LIN {X 0,Y 568.212,Z 444.708,A -85,B 0,C 180,E1 26844.426,E2 26844.426} C_VEL
LIN {X 0,Y 568.197,Z 444.71,A -85,B 0,C 180,E1 26841.145,E2 26841.145} C_VEL
LIN {X 0,Y 568.223,Z 444.707,A -85,B 0,C 180,E1 26837.829,E2 26837.829} C_VEL
LIN {X 0,Y 568.203,Z 444.709,A -85,B 0,C 180,E1 26834.47,E2 26834.47} C_VEL
LIN {X 0,Y 568.196,Z 444.71,A -85,B 0,C 180,E1 26831.161,E2 26831.161} C_VEL
LIN {X 0,Y 568.216,Z 444.708,A -85,B 0,C 180,E1 26827.889,E2 26827.889} C_VEL
LIN {X 0,Y 568.195,Z 444.71,A -85,B 0,C 180,E1 26824.542,E2 26824.542} C_VEL
LIN {X 0,Y 568.224,Z 444.705,A -85,B 0,C 180,E1 26821.21,E2 26821.21} C_VEL
LIN {X 0,Y 568.204,Z 444.708,A -85,B 0,C 180,E1 26817.882,E2 26817.882} C_VEL
LIN {X 0,Y 568.202,Z 444.709,A -85,B 0,C 180,E1 26814.648,E2 26814.648} C_VEL
LIN {X 0,Y 568.219,Z 444.706,A -85,B 0,C 180,E1 26811.398,E2 26811.398} C_VEL
LIN {X 0,Y 568.207,Z 444.707,A -85,B 0,C 180,E1 26808.061,E2 26808.061} C_VEL
LIN {X 0,Y 568.224,Z 444.706,A -85,B 0,C 180,E1 26804.636,E2 26804.636} C_VEL
LIN {X 0,Y 568.207,Z 444.707,A -85,B 0,C 180,E1 26801.321,E2 26801.321} C_VEL
LIN {X 0,Y 568.208,Z 444.71,A -85,B 0,C 180,E1 26799.787,E2 26799.787} C_VEL
LIN {X 0,Y 567.184,Z 444.832,A -85,B 0,C 180,E1 26799.011,E2 26799.011} C_VEL
LIN {X 0,Y 560.815,Z 445.632,A -85,B 0,C 180,E1 26796.831,E2 26796.831} C_VEL
LIN {X 0,Y 560.283,Z 445.694,A -85,B 0,C 180,E1 26796.264,E2 26796.264} C_VEL
LIN {X 0,Y 560.263,Z 445.695,A -85,B 0,C 180,E1 26792.93,E2 26792.93} C_VEL
LIN {X 0,Y 560.252,Z 445.696,A -85,B 0,C 180,E1 26789.665,E2 26789.665} C_VEL
LIN {X 0,Y 560.278,Z 445.695,A -85,B 0,C 180,E1 26786.412,E2 26786.412} C_VEL
LIN {X 0,Y 560.262,Z 445.697,A -85,B 0,C 180,E1 26783.083,E2 26783.083} C_VEL
LIN {X 0,Y 560.286,Z 445.693,A -85,B 0,C 180,E1 26779.759,E2 26779.759} C_VEL
LIN {X 0,Y 560.269,Z 445.697,A -85,B 0,C 180,E1 26776.431,E2 26776.431} C_VEL
LIN {X 0,Y 560.255,Z 445.701,A -85,B 0,C 180,E1 26773.119,E2 26773.119} C_VEL
LIN {X 0,Y 560.278,Z 445.696,A -85,B 0,C 180,E1 26769.882,E2 26769.882} C_VEL
LIN {X 0,Y 560.269,Z 445.7,A -85,B 0,C 180,E1 26766.575,E2 26766.575} C_VEL
LIN {X 0,Y 560.238,Z 445.797,A -85,B 0,C 180,E1 26764.175,E2 26764.175} C_VEL
LIN {X 0,Y 564.833,Z 458.966,A -85,B 0,C 180,E1 26762.797,E2 26762.797} C_VEL
LIN {X 0,Y 564.124,Z 495.402,A -85,B 0,C 180,E1 26759.984,E2 26759.984} C_VEL
LIN {X 0,Y 565.707,Z 504.661,A -85,B 0,C 180,E1 26759.758,E2 26759.758} C_VEL
LIN {X 0,Y 564.489,Z 747.125,A -85,B 0,C 180,E1 26756.4,E2 26756.4} C_VEL
LIN {X 0,Y 564.25,Z 768.15,A -85,B 0,C 180,E1 26755.998,E2 26755.998} C_VEL
LIN {X 0,Y 563.894,Z 788.378,A -85,B 0,C 180,E1 26755.42,E2 26755.42} C_VEL
LIN {X 0,Y 563.454,Z 808.539,A -85,B 0,C 180,E1 26754.645,E2 26754.645} C_VEL
LIN {X 0,Y 562.959,Z 828.494,A -85,B 0,C 180,E1 26753.665,E2 26753.665} C_VEL
LIN {X 0,Y 562.466,Z 847.374,A -85,B 0,C 180,E1 26752.519,E2 26752.519} C_VEL
LIN {X 0,Y 561.985,Z 864.434,A -85,B 0,C 180,E1 26751.281,E2 26751.281} C_VEL
LIN {X 0,Y 561.503,Z 881.299,A -85,B 0,C 180,E1 26749.829,E2 26749.829} C_VEL
LIN {X 0,Y 561.07,Z 897.052,A -85,B 0,C 180,E1 26748.224,E2 26748.224} C_VEL
LIN {X 0,Y 560.702,Z 911.608,A -85,B 0,C 180,E1 26746.471,E2 26746.471} C_VEL
LIN {X 0,Y 560.418,Z 924.193,A -85,B 0,C 180,E1 26744.675,E2 26744.675} C_VEL
LIN {X 0,Y 560.211,Z 935.329,A -85,B 0,C 180,E1 26742.786,E2 26742.786} C_VEL
LIN {X 0,Y 560.059,Z 944.99,A -85,B 0,C 180,E1 26740.804,E2 26740.804} C_VEL
LIN {X 0,Y 559.979,Z 953.12,A -85,B 0,C 180,E1 26738.729,E2 26738.729} C_VEL
LIN {X 0,Y 559.94,Z 959.122,A -85,B 0,C 180,E1 26736.768,E2 26736.768} C_VEL
LIN {X 0,Y 559.919,Z 963.693,A -85,B 0,C 180,E1 26734.711,E2 26734.711} C_VEL
LIN {X 0,Y 559.912,Z 966.567,A -85,B 0,C 180,E1 26732.661,E2 26732.661} C_VEL
LIN {X 0,Y 559.902,Z 967.886,A -85,B 0,C 180,E1 26730.511,E2 26730.511} C_VEL
LIN {X 0,Y 559.901,Z 967.469,A -85,B 0,C 180,E1 26728.362,E2 26728.362} C_VEL
LIN {X 0,Y 559.908,Z 965.467,A -85,B 0,C 180,E1 26726.314,E2 26726.314} C_VEL
LIN {X 0,Y 559.924,Z 961.822,A -85,B 0,C 180,E1 26724.26,E2 26724.26} C_VEL
LIN {X 0,Y 559.958,Z 956.427,A -85,B 0,C 180,E1 26722.2,E2 26722.2} C_VEL
LIN {X 0,Y 560.011,Z 949.242,A -85,B 0,C 180,E1 26720.13,E2 26720.13} C_VEL
LIN {X 0,Y 560.118,Z 940.592,A -85,B 0,C 180,E1 26718.153,E2 26718.153} C_VEL
LIN {X 0,Y 560.29,Z 930.551,A -85,B 0,C 180,E1 26716.27,E2 26716.27} C_VEL
LIN {X 0,Y 560.546,Z 918.433,A -85,B 0,C 180,E1 26714.374,E2 26714.374} C_VEL
LIN {X 0,Y 560.872,Z 904.72,A -85,B 0,C 180,E1 26712.572,E2 26712.572} C_VEL
LIN {X 0,Y 561.284,Z 889.331,A -85,B 0,C 180,E1 26710.866,E2 26710.866} C_VEL
LIN {X 0,Y 561.752,Z 872.597,A -85,B 0,C 180,E1 26709.3,E2 26709.3} C_VEL
LIN {X 0,Y 562.239,Z 855.595,A -85,B 0,C 180,E1 26707.961,E2 26707.961} C_VEL
LIN {X 0,Y 562.736,Z 837.569,A -85,B 0,C 180,E1 26706.768,E2 26706.768} C_VEL
LIN {X 0,Y 563.217,Z 818.644,A -85,B 0,C 180,E1 26705.733,E2 26705.733} C_VEL
LIN {X 0,Y 563.681,Z 798.675,A -85,B 0,C 180,E1 26704.86,E2 26704.86} C_VEL
LIN {X 0,Y 564.083,Z 778.165,A -85,B 0,C 180,E1 26704.174,E2 26704.174} C_VEL
LIN {X 0,Y 564.386,Z 757.733,A -85,B 0,C 180,E1 26703.688,E2 26703.688} C_VEL
LIN {X 0,Y 564.677,Z 708.736,A -85,B 0,C 180,E1 26702.983,E2 26702.983} C_VEL
LIN {X 0,Y 565.566,Z 507.584,A -85,B 0,C 180,E1 26700.186,E2 26700.186} C_VEL
LIN {X 0,Y 562.933,Z 497.494,A -85,B 0,C 180,E1 26699.882,E2 26699.882} C_VEL
LIN {X 0,Y 563.492,Z 471.301,A -85,B 0,C 180,E1 26696.81,E2 26696.81} C_VEL
LIN {X 0,Y 563.723,Z 457.22,A -85,B 0,C 180,E1 26695.118,E2 26695.118} C_VEL
LIN {X 0,Y 560.258,Z 445.701,A -85,B 0,C 180,E1 26693.474,E2 26693.474} C_VEL
LIN {X 0,Y 560.243,Z 445.699,A -85,B 0,C 180,E1 26690.123,E2 26690.123} C_VEL
LIN {X 0,Y 560.278,Z 445.693,A -85,B 0,C 180,E1 26686.878,E2 26686.878} C_VEL
LIN {X 0,Y 560.261,Z 445.695,A -85,B 0,C 180,E1 26683.541,E2 26683.541} C_VEL
LIN {X 0,Y 560.269,Z 445.691,A -85,B 0,C 180,E1 26680.109,E2 26680.109} C_VEL
LIN {X 0,Y 560.268,Z 445.697,A -85,B 0,C 180,E1 26676.843,E2 26676.843} C_VEL
LIN {X 0,Y 560.272,Z 445.699,A -85,B 0,C 180,E1 26673.466,E2 26673.466} C_VEL
LIN {X 0,Y 560.282,Z 445.696,A -85,B 0,C 180,E1 26670.058,E2 26670.058} C_VEL
LIN {X 0,Y 560.296,Z 445.883,A -85,B 0,C 180,E1 26668.994,E2 26668.994} C_VEL
LIN {X 0,Y 564.194,Z 457.95,A -85,B 0,C 180,E1 26667.551,E2 26667.551} C_VEL
LIN {X 0,Y 563.64,Z 489.328,A -85,B 0,C 180,E1 26664.582,E2 26664.582} C_VEL
LIN {X 0,Y 562.831,Z 522.784,A -85,B 0,C 180,E1 26661.467,E2 26661.467} C_VEL
LIN {X 0,Y 562.016,Z 560.717,A -85,B 0,C 180,E1 26657.979,E2 26657.979} C_VEL
LIN {X 0,Y 561.307,Z 595.844,A -85,B 0,C 180,E1 26654.758,E2 26654.758} C_VEL
LIN {X 0,Y 561.234,Z 603.069,A -85,B 0,C 180,E1 26654.135,E2 26654.135} C_VEL
LIN {X 0,Y 561.827,Z 610.203,A -85,B 0,C 180,E1 26654.019,E2 26654.019} C_VEL
LIN {X 0,Y 561.418,Z 743.182,A -85,B 0,C 180,E1 26652.262,E2 26652.262} C_VEL
LIN {X 0,Y 561.293,Z 759.345,A -85,B 0,C 180,E1 26651.88,E2 26651.88} C_VEL
LIN {X 0,Y 561.125,Z 773.652,A -85,B 0,C 180,E1 26651.356,E2 26651.356} C_VEL
LIN {X 0,Y 560.927,Z 786.575,A -85,B 0,C 180,E1 26650.735,E2 26650.735} C_VEL
LIN {X 0,Y 560.744,Z 799.431,A -85,B 0,C 180,E1 26649.96,E2 26649.96} C_VEL
LIN {X 0,Y 560.515,Z 813.552,A -85,B 0,C 180,E1 26648.876,E2 26648.876} C_VEL
LIN {X 0,Y 560.345,Z 823.86,A -85,B 0,C 180,E1 26647.897,E2 26647.897} C_VEL
LIN {X 0,Y 560.199,Z 833.784,A -85,B 0,C 180,E1 26646.765,E2 26646.765} C_VEL
LIN {X 0,Y 560.07,Z 843.961,A -85,B 0,C 180,E1 26645.327,E2 26645.327} C_VEL
LIN {X 0,Y 559.99,Z 851.364,A -85,B 0,C 180,E1 26643.993,E2 26643.993} C_VEL
LIN {X 0,Y 559.947,Z 857.668,A -85,B 0,C 180,E1 26642.559,E2 26642.559} C_VEL
LIN {X 0,Y 559.924,Z 863.148,A -85,B 0,C 180,E1 26640.819,E2 26640.819} C_VEL
LIN {X 0,Y 559.915,Z 866.195,A -85,B 0,C 180,E1 26639.284,E2 26639.284} C_VEL
LIN {X 0,Y 559.913,Z 867.841,A -85,B 0,C 180,E1 26637.646,E2 26637.646} C_VEL
LIN {X 0,Y 559.913,Z 867.666,A -85,B 0,C 180,E1 26636.007,E2 26636.007} C_VEL
LIN {X 0,Y 559.918,Z 865.949,A -85,B 0,C 180,E1 26634.467,E2 26634.467} C_VEL
LIN {X 0,Y 559.923,Z 862.739,A -85,B 0,C 180,E1 26632.923,E2 26632.923} C_VEL
LIN {X 0,Y 559.947,Z 857.342,A -85,B 0,C 180,E1 26631.27,E2 26631.27} C_VEL
LIN {X 0,Y 559.991,Z 851.393,A -85,B 0,C 180,E1 26629.923,E2 26629.923} C_VEL
LIN {X 0,Y 560.083,Z 843.245,A -85,B 0,C 180,E1 26628.467,E2 26628.467} C_VEL
LIN {X 0,Y 560.202,Z 833.489,A -85,B 0,C 180,E1 26627.109,E2 26627.109} C_VEL
LIN {X 0,Y 560.345,Z 823.82,A -85,B 0,C 180,E1 26626.008,E2 26626.008} C_VEL
LIN {X 0,Y 560.545,Z 812.105,A -85,B 0,C 180,E1 26624.905,E2 26624.905} C_VEL
LIN {X 0,Y 560.748,Z 798.703,A -85,B 0,C 180,E1 26623.903,E2 26623.903} C_VEL
LIN {X 0,Y 560.936,Z 786.019,A -85,B 0,C 180,E1 26623.145,E2 26623.145} C_VEL
LIN {X 0,Y 561.137,Z 773.052,A -85,B 0,C 180,E1 26622.528,E2 26622.528} C_VEL
LIN {X 0,Y 561.312,Z 756.063,A -85,B 0,C 180,E1 26621.941,E2 26621.941} C_VEL
LIN {X 0,Y 561.419,Z 741.983,A -85,B 0,C 180,E1 26621.627,E2 26621.627} C_VEL
LIN {X 0,Y 561.632,Z 605.827,A -85,B 0,C 180,E1 26619.816,E2 26619.816} C_VEL
LIN {X 0,Y 561.436,Z 603.897,A -85,B 0,C 180,E1 26619.761,E2 26619.761} C_VEL
LIN {X 0,Y 562.877,Z 569.056,A -85,B 0,C 180,E1 26616.387,E2 26616.387} C_VEL
LIN {X 0,Y 564.91,Z 533.555,A -85,B 0,C 180,E1 26612.829,E2 26612.829} C_VEL
LIN {X 0,Y 567.601,Z 501.05,A -85,B 0,C 180,E1 26609.397,E2 26609.397} C_VEL
LIN {X 0,Y 569.345,Z 484.628,A -85,B 0,C 180,E1 26607.554,E2 26607.554} C_VEL
LIN {X 0,Y 570.786,Z 468.2,A -85,B 0,C 180,E1 26605.475,E2 26605.475} C_VEL
LIN {X 0,Y 568.716,Z 463.182,A -85,B 0,C 180,E1 26604.29,E2 26604.29} C_VEL
LIN {X 0,Y 567.301,Z 459.69,A -85,B 0,C 180,E1 26603.31,E2 26603.31} C_VEL
LIN {X 0,Y 565.739,Z 455.845,A -85,B 0,C 180,E1 26601.858,E2 26601.858} C_VEL
LIN {X 0,Y 564.732,Z 454.619,A -85,B 0,C 180,E1 26600.529,E2 26600.529} C_VEL
LIN {X 0,Y 564.984,Z 454.894,A -85,B 0,C 180,E1 26599.364,E2 26599.364} C_VEL
LIN {X 0,Y 566.259,Z 456.589,A -85,B 0,C 180,E1 26598.324,E2 26598.324} C_VEL
LIN {X 0,Y 567.907,Z 460.494,A -85,B 0,C 180,E1 26597.326,E2 26597.326} C_VEL
LIN {X 0,Y 569.112,Z 464.051,A -85,B 0,C 180,E1 26596.71,E2 26596.71} C_VEL
LIN {X 0,Y 566.813,Z 482.57,A -85,B 0,C 180,E1 26595.237,E2 26595.237} C_VEL
LIN {X 0,Y 564.922,Z 510.213,A -85,B 0,C 180,E1 26593.302,E2 26593.302} C_VEL
LIN {X 0,Y 564.287,Z 540.963,A -85,B 0,C 180,E1 26591.298,E2 26591.298} C_VEL
LIN {X 0,Y 565.775,Z 557.767,A -85,B 0,C 180,E1 26590.169,E2 26590.169} C_VEL
LIN {X 0,Y 568.608,Z 569.698,A -85,B 0,C 180,E1 26589.312,E2 26589.312} C_VEL
LIN {X 0,Y 572.485,Z 578.868,A -85,B 0,C 180,E1 26588.596,E2 26588.596} C_VEL
LIN {X 0,Y 577.865,Z 586.598,A -85,B 0,C 180,E1 26587.908,E2 26587.908} C_VEL
LIN {X 0,Y 583.498,Z 591.893,A -85,B 0,C 180,E1 26587.336,E2 26587.336} C_VEL
LIN {X 0,Y 587.347,Z 594.24,A -85,B 0,C 180,E1 26586.861,E2 26586.861} C_VEL
LIN {X 0,Y 590.651,Z 595.228,A -85,B 0,C 180,E1 26586.315,E2 26586.315} C_VEL
LIN {X 0,Y 592.846,Z 594.931,A -85,B 0,C 180,E1 26585.784,E2 26585.784} C_VEL
LIN {X 0,Y 594.074,Z 593.569,A -85,B 0,C 180,E1 26585.261,E2 26585.261} C_VEL
LIN {X 0,Y 594.221,Z 590.934,A -85,B 0,C 180,E1 26584.692,E2 26584.692} C_VEL
LIN {X 0,Y 592.942,Z 587.105,A -85,B 0,C 180,E1 26584.162,E2 26584.162} C_VEL
LIN {X 0,Y 589.902,Z 581.364,A -85,B 0,C 180,E1 26583.66,E2 26583.66} C_VEL
LIN {X 0,Y 586.325,Z 572.675,A -85,B 0,C 180,E1 26583.131,E2 26583.131} C_VEL
LIN {X 0,Y 583.607,Z 562.507,A -85,B 0,C 180,E1 26582.72,E2 26582.72} C_VEL
LIN {X 0,Y 581.84,Z 551.15,A -85,B 0,C 180,E1 26582.448,E2 26582.448} C_VEL
LIN {X 0,Y 580.983,Z 537.863,A -85,B 0,C 180,E1 26582.315,E2 26582.315} C_VEL
LIN {X 0,Y 580.854,Z 522.497,A -85,B 0,C 180,E1 26582.295,E2 26582.295} C_VEL
LIN {X 0,Y 577.341,Z 528.82,A -85,B 0,C 180,E1 26581.739,E2 26581.739} C_VEL
LIN {X 0,Y 574.597,Z 531.681,A -85,B 0,C 180,E1 26581.294,E2 26581.294} C_VEL
LIN {X 0,Y 569.784,Z 544.591,A -85,B 0,C 180,E1 26580.489,E2 26580.489} C_VEL
LIN {X 0,Y 568.425,Z 548.114,A -85,B 0,C 180,E1 26580.255,E2 26580.255} C_VEL
LIN {X 0,Y 567.076,Z 552.625,A -85,B 0,C 180,E1 26580.021,E2 26580.021} C_VEL
LIN {X 0,Y 565.954,Z 557.205,A -85,B 0,C 180,E1 26579.823,E2 26579.823} C_VEL
LIN {X 0,Y 565.633,Z 557.842,A -85,B 0,C 180,E1 26579.762,E2 26579.762} C_VEL
LIN {X 0,Y 564.41,Z 806.369,A -85,B 0,C 180,E1 26576.292,E2 26576.292} C_VEL
LIN {X 0,Y 564.094,Z 827.689,A -85,B 0,C 180,E1 26575.795,E2 26575.795} C_VEL
LIN {X 0,Y 563.708,Z 847.582,A -85,B 0,C 180,E1 26575.139,E2 26575.139} C_VEL
LIN {X 0,Y 563.277,Z 866.639,A -85,B 0,C 180,E1 26574.32,E2 26574.32} C_VEL
LIN {X 0,Y 562.788,Z 885.877,A -85,B 0,C 180,E1 26573.291,E2 26573.291} C_VEL
LIN {X 0,Y 562.289,Z 903.978,A -85,B 0,C 180,E1 26572.114,E2 26572.114} C_VEL
LIN {X 0,Y 561.774,Z 921.539,A -85,B 0,C 180,E1 26570.744,E2 26570.744} C_VEL
LIN {X 0,Y 561.289,Z 938.854,A -85,B 0,C 180,E1 26569.134,E2 26569.134} C_VEL
LIN {X 0,Y 560.896,Z 953.414,A -85,B 0,C 180,E1 26567.534,E2 26567.534} C_VEL
LIN {X 0,Y 560.564,Z 967.357,A -85,B 0,C 180,E1 26565.731,E2 26565.731} C_VEL
LIN {X 0,Y 560.314,Z 979.299,A -85,B 0,C 180,E1 26563.893,E2 26563.893} C_VEL
LIN {X 0,Y 560.132,Z 989.854,A -85,B 0,C 180,E1 26561.951,E2 26561.951} C_VEL
LIN {X 0,Y 560.016,Z 998.675,A -85,B 0,C 180,E1 26559.974,E2 26559.974} C_VEL
LIN {X 0,Y 559.958,Z 1005.979,A -85,B 0,C 180,E1 26557.903,E2 26557.903} C_VEL
LIN {X 0,Y 559.93,Z 1011.245,A -85,B 0,C 180,E1 26555.944,E2 26555.944} C_VEL
LIN {X 0,Y 559.915,Z 1015.258,A -85,B 0,C 180,E1 26553.789,E2 26553.789} C_VEL
LIN {X 0,Y 559.907,Z 1017.386,A -85,B 0,C 180,E1 26551.74,E2 26551.74} C_VEL
LIN {X 0,Y 559.9,Z 1017.918,A -85,B 0,C 180,E1 26549.591,E2 26549.591} C_VEL
LIN {X 0,Y 559.907,Z 1016.847,A -85,B 0,C 180,E1 26547.544,E2 26547.544} C_VEL
LIN {X 0,Y 559.917,Z 1013.957,A -85,B 0,C 180,E1 26545.391,E2 26545.391} C_VEL
LIN {X 0,Y 559.937,Z 1009.727,A -85,B 0,C 180,E1 26543.438,E2 26543.438} C_VEL
LIN {X 0,Y 559.979,Z 1003.64,A -85,B 0,C 180,E1 26541.375,E2 26541.375} C_VEL
LIN {X 0,Y 560.052,Z 996.107,A -85,B 0,C 180,E1 26539.404,E2 26539.404} C_VEL
LIN {X 0,Y 560.195,Z 986.708,A -85,B 0,C 180,E1 26537.424,E2 26537.424} C_VEL
LIN {X 0,Y 560.381,Z 975.799,A -85,B 0,C 180,E1 26535.535,E2 26535.535} C_VEL
LIN {X 0,Y 560.681,Z 962.62,A -85,B 0,C 180,E1 26533.619,E2 26533.619} C_VEL
LIN {X 0,Y 561.017,Z 948.816,A -85,B 0,C 180,E1 26531.935,E2 26531.935} C_VEL
LIN {X 0,Y 561.46,Z 932.865,A -85,B 0,C 180,E1 26530.278,E2 26530.278} C_VEL
LIN {X 0,Y 561.94,Z 916.056,A -85,B 0,C 180,E1 26528.804,E2 26528.804} C_VEL
LIN {X 0,Y 562.446,Z 898.096,A -85,B 0,C 180,E1 26527.482,E2 26527.482} C_VEL
LIN {X 0,Y 562.937,Z 879.326,A -85,B 0,C 180,E1 26526.334,E2 26526.334} C_VEL
LIN {X 0,Y 563.439,Z 859.599,A -85,B 0,C 180,E1 26525.354,E2 26525.354} C_VEL
LIN {X 0,Y 563.895,Z 839.169,A -85,B 0,C 180,E1 26524.559,E2 26524.559} C_VEL
LIN {X 0,Y 564.243,Z 818.543,A -85,B 0,C 180,E1 26523.966,E2 26523.966} C_VEL
LIN {X 0,Y 564.48,Z 797.161,A -85,B 0,C 180,E1 26523.557,E2 26523.557} C_VEL
LIN {X 0,Y 565.701,Z 557.499,A -85,B 0,C 180,E1 26520.221,E2 26520.221} C_VEL
LIN {X 0,Y 566.509,Z 555.474,A -85,B 0,C 180,E1 26520.079,E2 26520.079} C_VEL
LIN {X 0,Y 567.509,Z 551.007,A -85,B 0,C 180,E1 26519.904,E2 26519.904} C_VEL
LIN {X 0,Y 569.272,Z 545.742,A -85,B 0,C 180,E1 26519.599,E2 26519.599} C_VEL
LIN {X 0,Y 573.361,Z 535.153,A -85,B 0,C 180,E1 26518.91,E2 26518.91} C_VEL
LIN {X 0,Y 574.591,Z 531.68,A -85,B 0,C 180,E1 26518.707,E2 26518.707} C_VEL
LIN {X 0,Y 577.335,Z 528.827,A -85,B 0,C 180,E1 26518.262,E2 26518.262} C_VEL
LIN {X 0,Y 580.897,Z 522.403,A -85,B 0,C 180,E1 26517.698,E2 26517.698} C_VEL
LIN {X 0,Y 581.148,Z 542.214,A -85,B 0,C 180,E1 26517.659,E2 26517.659} C_VEL
LIN {X 0,Y 582.272,Z 554.667,A -85,B 0,C 180,E1 26517.485,E2 26517.485} C_VEL
LIN {X 0,Y 584.278,Z 565.498,A -85,B 0,C 180,E1 26517.178,E2 26517.178} C_VEL
LIN {X 0,Y 587.14,Z 574.973,A -85,B 0,C 180,E1 26516.747,E2 26516.747} C_VEL
LIN {X 0,Y 590.798,Z 583.078,A -85,B 0,C 180,E1 26516.21,E2 26516.21} C_VEL
LIN {X 0,Y 593.208,Z 587.704,A -85,B 0,C 180,E1 26515.769,E2 26515.769} C_VEL
LIN {X 0,Y 594.283,Z 591.409,A -85,B 0,C 180,E1 26515.226,E2 26515.226} C_VEL
LIN {X 0,Y 594.044,Z 593.64,A -85,B 0,C 180,E1 26514.718,E2 26514.718} C_VEL
LIN {X 0,Y 592.459,Z 595.083,A -85,B 0,C 180,E1 26514.102,E2 26514.102} C_VEL
LIN {X 0,Y 589.617,Z 595.055,A -85,B 0,C 180,E1 26513.494,E2 26513.494} C_VEL
LIN {X 0,Y 586.119,Z 593.612,A -85,B 0,C 180,E1 26512.973,E2 26512.973} C_VEL
LIN {X 0,Y 580.24,Z 589.13,A -85,B 0,C 180,E1 26512.273,E2 26512.273} C_VEL
LIN {X 0,Y 575.058,Z 582.688,A -85,B 0,C 180,E1 26511.505,E2 26511.505} C_VEL
LIN {X 0,Y 571.39,Z 575.079,A -85,B 0,C 180,E1 26510.743,E2 26510.743} C_VEL
LIN {X 0,Y 568.573,Z 564.258,A -85,B 0,C 180,E1 26509.806,E2 26509.806} C_VEL
LIN {X 0,Y 567.205,Z 550.519,A -85,B 0,C 180,E1 26508.756,E2 26508.756} C_VEL
LIN {X 0,Y 568.262,Z 497.326,A -85,B 0,C 180,E1 26504.983,E2 26504.983} C_VEL
LIN {X 0,Y 569.217,Z 464.903,A -85,B 0,C 180,E1 26502.585,E2 26502.585} C_VEL
LIN {X 0,Y 561.938,Z 449.676,A -85,B 0,C 180,E1 26500.634,E2 26500.634} C_VEL
LIN {X 0,Y 560.368,Z 446.244,A -85,B 0,C 180,E1 26500.187,E2 26500.187} C_VEL
LIN {X 0,Y 560.28,Z 445.7,A -85,B 0,C 180,E1 26500.108,E2 26500.108} C_VEL
LIN {X 0,Y 560.229,Z 445.698,A -85,B 0,C 180,E1 26496.913,E2 26496.913} C_VEL
LIN {X 0,Y 560.258,Z 445.696,A -85,B 0,C 180,E1 26493.549,E2 26493.549} C_VEL
LIN {X 0,Y 560.259,Z 445.696,A -85,B 0,C 180,E1 26490.335,E2 26490.335} C_VEL
LIN {X 0,Y 560.233,Z 445.699,A -85,B 0,C 180,E1 26486.957,E2 26486.957} C_VEL
LIN {X 0,Y 560.28,Z 445.693,A -85,B 0,C 180,E1 26483.674,E2 26483.674} C_VEL
LIN {X 0,Y 560.225,Z 445.699,A -85,B 0,C 180,E1 26480.449,E2 26480.449} C_VEL
LIN {X 0,Y 560.255,Z 445.696,A -85,B 0,C 180,E1 26477.018,E2 26477.018} C_VEL
LIN {X 0,Y 560.257,Z 445.696,A -85,B 0,C 180,E1 26473.836,E2 26473.836} C_VEL
LIN {X 0,Y 560.227,Z 445.699,A -85,B 0,C 180,E1 26470.46,E2 26470.46} C_VEL
LIN {X 0,Y 560.281,Z 445.692,A -85,B 0,C 180,E1 26467.156,E2 26467.156} C_VEL
LIN {X 0,Y 560.225,Z 445.699,A -85,B 0,C 180,E1 26463.918,E2 26463.918} C_VEL
LIN {X 0,Y 560.253,Z 445.695,A -85,B 0,C 180,E1 26460.511,E2 26460.511} C_VEL
LIN {X 0,Y 560.256,Z 445.695,A -85,B 0,C 180,E1 26457.34,E2 26457.34} C_VEL
LIN {X 0,Y 560.225,Z 445.698,A -85,B 0,C 180,E1 26453.955,E2 26453.955} C_VEL
LIN {X 0,Y 560.279,Z 445.691,A -85,B 0,C 180,E1 26450.701,E2 26450.701} C_VEL
LIN {X 0,Y 560.228,Z 445.695,A -85,B 0,C 180,E1 26447.424,E2 26447.424} C_VEL
LIN {X 0,Y 560.251,Z 445.696,A -85,B 0,C 180,E1 26443.941,E2 26443.941} C_VEL
LIN {X 0,Y 560.26,Z 445.693,A -85,B 0,C 180,E1 26440.722,E2 26440.722} C_VEL
LIN {X 0,Y 560.225,Z 445.694,A -85,B 0,C 180,E1 26437.324,E2 26437.324} C_VEL
LIN {X 0,Y 560.283,Z 445.694,A -85,B 0,C 180,E1 26436.264,E2 26436.264} C_VEL
LIN {X 0,Y 559.284,Z 445.817,A -85,B 0,C 180,E1 26435.476,E2 26435.476} C_VEL
LIN {X 0,Y 552.853,Z 446.619,A -85,B 0,C 180,E1 26433.265,E2 26433.265} C_VEL
LIN {X 0,Y 552.32,Z 446.682,A -85,B 0,C 180,E1 26432.689,E2 26432.689} C_VEL
LIN {X 0,Y 552.289,Z 446.685,A -85,B 0,C 180,E1 26429.301,E2 26429.301} C_VEL
LIN {X 0,Y 552.339,Z 446.681,A -85,B 0,C 180,E1 26426.113,E2 26426.113} C_VEL
LIN {X 0,Y 552.301,Z 446.686,A -85,B 0,C 180,E1 26422.796,E2 26422.796} C_VEL
LIN {X 0,Y 552.328,Z 446.681,A -85,B 0,C 180,E1 26419.467,E2 26419.467} C_VEL
LIN {X 0,Y 552.323,Z 446.686,A -85,B 0,C 180,E1 26416.244,E2 26416.244} C_VEL
LIN {X 0,Y 552.298,Z 446.69,A -85,B 0,C 180,E1 26412.897,E2 26412.897} C_VEL
LIN {X 0,Y 552.339,Z 446.684,A -85,B 0,C 180,E1 26409.705,E2 26409.705} C_VEL
LIN {X 0,Y 552.307,Z 446.69,A -85,B 0,C 180,E1 26406.297,E2 26406.297} C_VEL
LIN {X 0,Y 552.311,Z 446.756,A -85,B 0,C 180,E1 26404.641,E2 26404.641} C_VEL
LIN {X 0,Y 557.679,Z 461.976,A -85,B 0,C 180,E1 26403.027,E2 26403.027} C_VEL
LIN {X 0,Y 556.92,Z 495.437,A -85,B 0,C 180,E1 26400.412,E2 26400.412} C_VEL
LIN {X 0,Y 558.758,Z 505.983,A -85,B 0,C 180,E1 26400.148,E2 26400.148} C_VEL
LIN {X 0,Y 557.305,Z 748.805,A -85,B 0,C 180,E1 26396.741,E2 26396.741} C_VEL
LIN {X 0,Y 557.019,Z 769.975,A -85,B 0,C 180,E1 26396.318,E2 26396.318} C_VEL
LIN {X 0,Y 556.593,Z 790.574,A -85,B 0,C 180,E1 26395.703,E2 26395.703} C_VEL
LIN {X 0,Y 556.085,Z 809.793,A -85,B 0,C 180,E1 26394.937,E2 26394.937} C_VEL
LIN {X 0,Y 555.518,Z 829.135,A -85,B 0,C 180,E1 26393.965,E2 26393.965} C_VEL
LIN {X 0,Y 554.928,Z 848.12,A -85,B 0,C 180,E1 26392.791,E2 26392.791} C_VEL
LIN {X 0,Y 554.335,Z 865.766,A -85,B 0,C 180,E1 26391.478,E2 26391.478} C_VEL
LIN {X 0,Y 553.789,Z 881.86,A -85,B 0,C 180,E1 26390.062,E2 26390.062} C_VEL
LIN {X 0,Y 553.279,Z 897.649,A -85,B 0,C 180,E1 26388.422,E2 26388.422} C_VEL
LIN {X 0,Y 552.857,Z 911.61,A -85,B 0,C 180,E1 26386.711,E2 26386.711} C_VEL
LIN {X 0,Y 552.524,Z 924.195,A -85,B 0,C 180,E1 26384.89,E2 26384.89} C_VEL
LIN {X 0,Y 552.274,Z 935.33,A -85,B 0,C 180,E1 26382.973,E2 26382.973} C_VEL
LIN {X 0,Y 552.093,Z 944.995,A -85,B 0,C 180,E1 26380.961,E2 26380.961} C_VEL
LIN {X 0,Y 551.989,Z 953.123,A -85,B 0,C 180,E1 26378.856,E2 26378.856} C_VEL
LIN {X 0,Y 551.94,Z 959.125,A -85,B 0,C 180,E1 26376.866,E2 26376.866} C_VEL
LIN {X 0,Y 551.92,Z 963.695,A -85,B 0,C 180,E1 26374.78,E2 26374.78} C_VEL
LIN {X 0,Y 551.913,Z 966.568,A -85,B 0,C 180,E1 26372.699,E2 26372.699} C_VEL
LIN {X 0,Y 551.902,Z 967.886,A -85,B 0,C 180,E1 26370.518,E2 26370.518} C_VEL
LIN {X 0,Y 551.902,Z 967.469,A -85,B 0,C 180,E1 26368.338,E2 26368.338} C_VEL
LIN {X 0,Y 551.91,Z 965.466,A -85,B 0,C 180,E1 26366.26,E2 26366.26} C_VEL
LIN {X 0,Y 551.929,Z 961.821,A -85,B 0,C 180,E1 26364.177,E2 26364.177} C_VEL
LIN {X 0,Y 551.965,Z 956.426,A -85,B 0,C 180,E1 26362.086,E2 26362.086} C_VEL
LIN {X 0,Y 552.033,Z 949.241,A -85,B 0,C 180,E1 26359.986,E2 26359.986} C_VEL
LIN {X 0,Y 552.177,Z 940.076,A -85,B 0,C 180,E1 26357.874,E2 26357.874} C_VEL
LIN {X 0,Y 552.401,Z 929.287,A -85,B 0,C 180,E1 26355.856,E2 26355.856} C_VEL
LIN {X 0,Y 552.709,Z 916.902,A -85,B 0,C 180,E1 26353.931,E2 26353.931} C_VEL
LIN {X 0,Y 553.087,Z 903.805,A -85,B 0,C 180,E1 26352.21,E2 26352.21} C_VEL
LIN {X 0,Y 553.568,Z 888.801,A -85,B 0,C 180,E1 26350.535,E2 26350.535} C_VEL
LIN {X 0,Y 554.12,Z 872.076,A -85,B 0,C 180,E1 26348.956,E2 26348.956} C_VEL
LIN {X 0,Y 554.734,Z 854.133,A -85,B 0,C 180,E1 26347.535,E2 26347.535} C_VEL
LIN {X 0,Y 555.33,Z 835.779,A -85,B 0,C 180,E1 26346.327,E2 26346.327} C_VEL
LIN {X 0,Y 555.905,Z 816.826,A -85,B 0,C 180,E1 26345.301,E2 26345.301} C_VEL
LIN {X 0,Y 556.431,Z 796.657,A -85,B 0,C 180,E1 26344.429,E2 26344.429} C_VEL
LIN {X 0,Y 556.882,Z 776.082,A -85,B 0,C 180,E1 26343.756,E2 26343.756} C_VEL
LIN {X 0,Y 557.241,Z 754.862,A -85,B 0,C 180,E1 26343.273,E2 26343.273} C_VEL
LIN {X 0,Y 558.655,Z 509.404,A -85,B 0,C 180,E1 26339.806,E2 26339.806} C_VEL
LIN {X 0,Y 555.492,Z 497.283,A -85,B 0,C 180,E1 26339.411,E2 26339.411} C_VEL
LIN {X 0,Y 556.167,Z 472.309,A -85,B 0,C 180,E1 26336.439,E2 26336.439} C_VEL
LIN {X 0,Y 556.32,Z 459.961,A -85,B 0,C 180,E1 26334.942,E2 26334.942} C_VEL
LIN {X 0,Y 552.345,Z 446.687,A -85,B 0,C 180,E1 26333.026,E2 26333.026} C_VEL
LIN {X 0,Y 552.307,Z 446.691,A -85,B 0,C 180,E1 26329.737,E2 26329.737} C_VEL
LIN {X 0,Y 552.331,Z 446.679,A -85,B 0,C 180,E1 26326.392,E2 26326.392} C_VEL
LIN {X 0,Y 552.338,Z 446.685,A -85,B 0,C 180,E1 26323.001,E2 26323.001} C_VEL
LIN {X 0,Y 552.322,Z 446.684,A -85,B 0,C 180,E1 26319.702,E2 26319.702} C_VEL
LIN {X 0,Y 552.337,Z 446.682,A -85,B 0,C 180,E1 26316.335,E2 26316.335} C_VEL
LIN {X 0,Y 552.328,Z 446.691,A -85,B 0,C 180,E1 26312.894,E2 26312.894} C_VEL
LIN {X 0,Y 552.337,Z 446.689,A -85,B 0,C 180,E1 26309.617,E2 26309.617} C_VEL
LIN {X 0,Y 552.358,Z 446.837,A -85,B 0,C 180,E1 26309.46,E2 26309.46} C_VEL
LIN {X 0,Y 556.965,Z 461.376,A -85,B 0,C 180,E1 26307.707,E2 26307.707} C_VEL
LIN {X 0,Y 556.279,Z 492.827,A -85,B 0,C 180,E1 26304.702,E2 26304.702} C_VEL
LIN {X 0,Y 555.415,Z 525.871,A -85,B 0,C 180,E1 26301.601,E2 26301.601} C_VEL
LIN {X 0,Y 554.516,Z 562.768,A -85,B 0,C 180,E1 26298.176,E2 26298.176} C_VEL
LIN {X 0,Y 553.783,Z 597.7,A -85,B 0,C 180,E1 26294.963,E2 26294.963} C_VEL
LIN {X 0,Y 553.726,Z 604.219,A -85,B 0,C 180,E1 26294.397,E2 26294.397} C_VEL
LIN {X 0,Y 554.281,Z 611.085,A -85,B 0,C 180,E1 26294.283,E2 26294.283} C_VEL
LIN {X 0,Y 553.721,Z 743.19,A -85,B 0,C 180,E1 26292.488,E2 26292.488} C_VEL
LIN {X 0,Y 553.59,Z 758.732,A -85,B 0,C 180,E1 26292.124,E2 26292.124} C_VEL
LIN {X 0,Y 553.382,Z 773.801,A -85,B 0,C 180,E1 26291.57,E2 26291.57} C_VEL
LIN {X 0,Y 553.143,Z 786.632,A -85,B 0,C 180,E1 26290.941,E2 26290.941} C_VEL
LIN {X 0,Y 552.92,Z 798.556,A -85,B 0,C 180,E1 26290.208,E2 26290.208} C_VEL
LIN {X 0,Y 552.646,Z 812.874,A -85,B 0,C 180,E1 26289.109,E2 26289.109} C_VEL
LIN {X 0,Y 552.438,Z 823.442,A -85,B 0,C 180,E1 26288.099,E2 26288.099} C_VEL
LIN {X 0,Y 552.276,Z 832.446,A -85,B 0,C 180,E1 26287.072,E2 26287.072} C_VEL
LIN {X 0,Y 552.136,Z 841.589,A -85,B 0,C 180,E1 26285.821,E2 26285.821} C_VEL
LIN {X 0,Y 552.017,Z 850.559,A -85,B 0,C 180,E1 26284.259,E2 26284.259} C_VEL
LIN {X 0,Y 551.959,Z 856.599,A -85,B 0,C 180,E1 26282.908,E2 26282.908} C_VEL
LIN {X 0,Y 551.931,Z 861.592,A -85,B 0,C 180,E1 26281.453,E2 26281.453} C_VEL
LIN {X 0,Y 551.918,Z 865.623,A -85,B 0,C 180,E1 26279.689,E2 26279.689} C_VEL
LIN {X 0,Y 551.913,Z 867.415,A -85,B 0,C 180,E1 26278.235,E2 26278.235} C_VEL
LIN {X 0,Y 551.915,Z 867.922,A -85,B 0,C 180,E1 26276.781,E2 26276.781} C_VEL
LIN {X 0,Y 551.914,Z 866.822,A -85,B 0,C 180,E1 26275.012,E2 26275.012} C_VEL
LIN {X 0,Y 551.921,Z 864.085,A -85,B 0,C 180,E1 26273.447,E2 26273.447} C_VEL
LIN {X 0,Y 551.936,Z 860.442,A -85,B 0,C 180,E1 26272.087,E2 26272.087} C_VEL
LIN {X 0,Y 551.979,Z 855.076,A -85,B 0,C 180,E1 26270.618,E2 26270.618} C_VEL
LIN {X 0,Y 552.057,Z 847.133,A -85,B 0,C 180,E1 26269.008,E2 26269.008} C_VEL
LIN {X 0,Y 552.164,Z 839.375,A -85,B 0,C 180,E1 26267.769,E2 26267.769} C_VEL
LIN {X 0,Y 552.311,Z 830.532,A -85,B 0,C 180,E1 26266.602,E2 26266.602} C_VEL
LIN {X 0,Y 552.539,Z 818.659,A -85,B 0,C 180,E1 26265.325,E2 26265.325} C_VEL
LIN {X 0,Y 552.753,Z 806.842,A -85,B 0,C 180,E1 26264.311,E2 26264.311} C_VEL
LIN {X 0,Y 552.995,Z 795.753,A -85,B 0,C 180,E1 26263.509,E2 26263.509} C_VEL
LIN {X 0,Y 553.271,Z 782.006,A -85,B 0,C 180,E1 26262.706,E2 26262.706} C_VEL
LIN {X 0,Y 553.491,Z 767.007,A -85,B 0,C 180,E1 26262.061,E2 26262.061} C_VEL
LIN {X 0,Y 553.636,Z 753.452,A -85,B 0,C 180,E1 26261.641,E2 26261.641} C_VEL
LIN {X 0,Y 553.765,Z 738.251,A -85,B 0,C 180,E1 26261.333,E2 26261.333} C_VEL
LIN {X 0,Y 554.312,Z 607.285,A -85,B 0,C 180,E1 26259.52,E2 26259.52} C_VEL
LIN {X 0,Y 554.305,Z 606.119,A -85,B 0,C 180,E1 26259.461,E2 26259.461} C_VEL
LIN {X 0,Y 555.866,Z 572.667,A -85,B 0,C 180,E1 26256.183,E2 26256.183} C_VEL
LIN {X 0,Y 558.037,Z 538.385,A -85,B 0,C 180,E1 26252.698,E2 26252.698} C_VEL
LIN {X 0,Y 561.079,Z 505.791,A -85,B 0,C 180,E1 26249.199,E2 26249.199} C_VEL
LIN {X 0,Y 563.19,Z 488.496,A -85,B 0,C 180,E1 26247.216,E2 26247.216} C_VEL
LIN {X 0,Y 564.919,Z 473.045,A -85,B 0,C 180,E1 26245.21,E2 26245.21} C_VEL
LIN {X 0,Y 562.856,Z 468.08,A -85,B 0,C 180,E1 26243.927,E2 26243.927} C_VEL
LIN {X 0,Y 561.925,Z 465.491,A -85,B 0,C 180,E1 26243.156,E2 26243.156} C_VEL
LIN {X 0,Y 560.64,Z 461.965,A -85,B 0,C 180,E1 26241.694,E2 26241.694} C_VEL
LIN {X 0,Y 559.953,Z 460.995,A -85,B 0,C 180,E1 26240.264,E2 26240.264} C_VEL
LIN {X 0,Y 560.523,Z 461.685,A -85,B 0,C 180,E1 26239.107,E2 26239.107} C_VEL
LIN {X 0,Y 561.36,Z 462.924,A -85,B 0,C 180,E1 26238.425,E2 26238.425} C_VEL
LIN {X 0,Y 562.789,Z 466.85,A -85,B 0,C 180,E1 26237.399,E2 26237.399} C_VEL
LIN {X 0,Y 563.276,Z 468.702,A -85,B 0,C 180,E1 26237.066,E2 26237.066} C_VEL
LIN {X 0,Y 560.539,Z 485.693,A -85,B 0,C 180,E1 26235.635,E2 26235.635} C_VEL
LIN {X 0,Y 558.254,Z 510.616,A -85,B 0,C 180,E1 26233.798,E2 26233.798} C_VEL
LIN {X 0,Y 557.115,Z 541.508,A -85,B 0,C 180,E1 26231.704,E2 26231.704} C_VEL
LIN {X 0,Y 558.431,Z 559.596,A -85,B 0,C 180,E1 26230.452,E2 26230.452} C_VEL
LIN {X 0,Y 561.228,Z 572.215,A -85,B 0,C 180,E1 26229.519,E2 26229.519} C_VEL
LIN {X 0,Y 565.227,Z 582.171,A -85,B 0,C 180,E1 26228.73,E2 26228.73} C_VEL
LIN {X 0,Y 570.816,Z 590.652,A -85,B 0,C 180,E1 26227.979,E2 26227.979} C_VEL
LIN {X 0,Y 577.199,Z 597.025,A -85,B 0,C 180,E1 26227.335,E2 26227.335} C_VEL
LIN {X 0,Y 582.28,Z 600.528,A -85,B 0,C 180,E1 26226.852,E2 26226.852} C_VEL
LIN {X 0,Y 586.091,Z 602.101,A -85,B 0,C 180,E1 26226.369,E2 26226.369} C_VEL
LIN {X 0,Y 589.281,Z 602.409,A -85,B 0,C 180,E1 26225.802,E2 26225.802} C_VEL
LIN {X 0,Y 591.359,Z 601.372,A -85,B 0,C 180,E1 26225.209,E2 26225.209} C_VEL
LIN {X 0,Y 592.116,Z 599.111,A -85,B 0,C 180,E1 26224.6,E2 26224.6} C_VEL
LIN {X 0,Y 591.38,Z 595.652,A -85,B 0,C 180,E1 26224.031,E2 26224.031} C_VEL
LIN {X 0,Y 589.21,Z 591.411,A -85,B 0,C 180,E1 26223.559,E2 26223.559} C_VEL
LIN {X 0,Y 584.894,Z 582.926,A -85,B 0,C 180,E1 26222.916,E2 26222.916} C_VEL
LIN {X 0,Y 581.522,Z 573.253,A -85,B 0,C 180,E1 26222.399,E2 26222.399} C_VEL
LIN {X 0,Y 579.024,Z 562.34,A -85,B 0,C 180,E1 26222.007,E2 26222.007} C_VEL
LIN {X 0,Y 577.407,Z 550.024,A -85,B 0,C 180,E1 26221.75,E2 26221.75} C_VEL
LIN {X 0,Y 576.751,Z 539.815,A -85,B 0,C 180,E1 26221.644,E2 26221.644} C_VEL
LIN {X 0,Y 572.401,Z 550.885,A -85,B 0,C 180,E1 26220.931,E2 26220.931} C_VEL
LIN {X 0,Y 570.578,Z 556.933,A -85,B 0,C 180,E1 26220.624,E2 26220.624} C_VEL
LIN {X 0,Y 569.388,Z 562.129,A -85,B 0,C 180,E1 26220.421,E2 26220.421} C_VEL
LIN {X 0,Y 565.179,Z 621.658,A -85,B 0,C 180,E1 26219.686,E2 26219.686} C_VEL
LIN {X 0,Y 561.533,Z 663.367,A -85,B 0,C 180,E1 26219.027,E2 26219.027} C_VEL
LIN {X 0,Y 559.274,Z 682.17,A -85,B 0,C 180,E1 26218.607,E2 26218.607} C_VEL
LIN {X 0,Y 558.23,Z 686.94,A -85,B 0,C 180,E1 26218.41,E2 26218.41} C_VEL
LIN {X 0,Y 557.888,Z 687.751,A -85,B 0,C 180,E1 26218.34,E2 26218.34} C_VEL
LIN {X 0,Y 557.229,Z 806.548,A -85,B 0,C 180,E1 26216.654,E2 26216.654} C_VEL
LIN {X 0,Y 556.858,Z 828.017,A -85,B 0,C 180,E1 26216.146,E2 26216.146} C_VEL
LIN {X 0,Y 556.399,Z 848.329,A -85,B 0,C 180,E1 26215.464,E2 26215.464} C_VEL
LIN {X 0,Y 555.876,Z 867.765,A -85,B 0,C 180,E1 26214.608,E2 26214.608} C_VEL
LIN {X 0,Y 555.3,Z 886.893,A -85,B 0,C 180,E1 26213.562,E2 26213.562} C_VEL
LIN {X 0,Y 554.702,Z 905.003,A -85,B 0,C 180,E1 26212.355,E2 26212.355} C_VEL
LIN {X 0,Y 554.114,Z 922.163,A -85,B 0,C 180,E1 26210.989,E2 26210.989} C_VEL
LIN {X 0,Y 553.54,Z 939.361,A -85,B 0,C 180,E1 26209.358,E2 26209.358} C_VEL
LIN {X 0,Y 553.096,Z 953.409,A -85,B 0,C 180,E1 26207.789,E2 26207.789} C_VEL
LIN {X 0,Y 552.698,Z 967.35,A -85,B 0,C 180,E1 26205.961,E2 26205.961} C_VEL
LIN {X 0,Y 552.407,Z 979.016,A -85,B 0,C 180,E1 26204.144,E2 26204.144} C_VEL
LIN {X 0,Y 552.179,Z 990.009,A -85,B 0,C 180,E1 26202.095,E2 26202.095} C_VEL
LIN {X 0,Y 552.034,Z 999.086,A -85,B 0,C 180,E1 26200.014,E2 26200.014} C_VEL
LIN {X 0,Y 551.965,Z 1006.286,A -85,B 0,C 180,E1 26197.914,E2 26197.914} C_VEL
LIN {X 0,Y 551.931,Z 1011.736,A -85,B 0,C 180,E1 26195.823,E2 26195.823} C_VEL
LIN {X 0,Y 551.908,Z 1015.537,A -85,B 0,C 180,E1 26193.636,E2 26193.636} C_VEL
LIN {X 0,Y 551.9,Z 1017.521,A -85,B 0,C 180,E1 26191.558,E2 26191.558} C_VEL
LIN {X 0,Y 551.902,Z 1017.874,A -85,B 0,C 180,E1 26189.378,E2 26189.378} C_VEL
LIN {X 0,Y 551.912,Z 1016.526,A -85,B 0,C 180,E1 26187.197,E2 26187.197} C_VEL
LIN {X 0,Y 551.919,Z 1013.564,A -85,B 0,C 180,E1 26185.116,E2 26185.116} C_VEL
LIN {X 0,Y 551.938,Z 1009.096,A -85,B 0,C 180,E1 26183.083,E2 26183.083} C_VEL
LIN {X 0,Y 551.991,Z 1002.575,A -85,B 0,C 180,E1 26180.934,E2 26180.934} C_VEL
LIN {X 0,Y 552.096,Z 994.742,A -85,B 0,C 180,E1 26178.933,E2 26178.933} C_VEL
LIN {X 0,Y 552.281,Z 984.898,A -85,B 0,C 180,E1 26176.906,E2 26176.906} C_VEL
LIN {X 0,Y 552.538,Z 973.826,A -85,B 0,C 180,E1 26175.004,E2 26175.004} C_VEL
LIN {X 0,Y 552.865,Z 961.093,A -85,B 0,C 180,E1 26173.181,E2 26173.181} C_VEL
LIN {X 0,Y 553.301,Z 946.962,A -85,B 0,C 180,E1 26171.456,E2 26171.456} C_VEL
LIN {X 0,Y 553.794,Z 931.447,A -85,B 0,C 180,E1 26169.858,E2 26169.858} C_VEL
LIN {X 0,Y 554.364,Z 914.985,A -85,B 0,C 180,E1 26168.412,E2 26168.412} C_VEL
LIN {X 0,Y 554.968,Z 897.194,A -85,B 0,C 180,E1 26167.099,E2 26167.099} C_VEL
LIN {X 0,Y 555.553,Z 878.34,A -85,B 0,C 180,E1 26165.944,E2 26165.944} C_VEL
LIN {X 0,Y 556.133,Z 858.366,A -85,B 0,C 180,E1 26164.951,E2 26164.951} C_VEL
LIN {X 0,Y 556.639,Z 838.145,A -85,B 0,C 180,E1 26164.169,E2 26164.169} C_VEL
LIN {X 0,Y 557.059,Z 817.518,A -85,B 0,C 180,E1 26163.579,E2 26163.579} C_VEL
LIN {X 0,Y 557.331,Z 796.163,A -85,B 0,C 180,E1 26163.175,E2 26163.175} C_VEL
LIN {X 0,Y 557.929,Z 687.343,A -85,B 0,C 180,E1 26161.648,E2 26161.648} C_VEL
LIN {X 0,Y 558.672,Z 685.439,A -85,B 0,C 180,E1 26161.507,E2 26161.507} C_VEL
LIN {X 0,Y 560.364,Z 674.075,A -85,B 0,C 180,E1 26161.189,E2 26161.189} C_VEL
LIN {X 0,Y 563.418,Z 643.096,A -85,B 0,C 180,E1 26160.63,E2 26160.63} C_VEL
LIN {X 0,Y 567.729,Z 587.176,A -85,B 0,C 180,E1 26159.866,E2 26159.866} C_VEL
LIN {X 0,Y 569.589,Z 560.911,A -85,B 0,C 180,E1 26159.545,E2 26159.545} C_VEL
LIN {X 0,Y 571.371,Z 554.062,A -85,B 0,C 180,E1 26159.242,E2 26159.242} C_VEL
LIN {X 0,Y 572.782,Z 550.043,A -85,B 0,C 180,E1 26159.006,E2 26159.006} C_VEL
LIN {X 0,Y 576.798,Z 539.845,A -85,B 0,C 180,E1 26158.348,E2 26158.348} C_VEL
LIN {X 0,Y 577.747,Z 553.413,A -85,B 0,C 180,E1 26158.196,E2 26158.196} C_VEL
LIN {X 0,Y 579.582,Z 565.261,A -85,B 0,C 180,E1 26157.904,E2 26157.904} C_VEL
LIN {X 0,Y 582.355,Z 576.016,A -85,B 0,C 180,E1 26157.472,E2 26157.472} C_VEL
LIN {X 0,Y 586.114,Z 585.665,A -85,B 0,C 180,E1 26156.9,E2 26156.9} C_VEL
LIN {X 0,Y 590.255,Z 593.236,A -85,B 0,C 180,E1 26156.262,E2 26156.262} C_VEL
LIN {X 0,Y 591.835,Z 597.031,A -85,B 0,C 180,E1 26155.766,E2 26155.766} C_VEL
LIN {X 0,Y 592.016,Z 600.04,A -85,B 0,C 180,E1 26155.191,E2 26155.191} C_VEL
LIN {X 0,Y 590.949,Z 601.751,A -85,B 0,C 180,E1 26154.639,E2 26154.639} C_VEL
LIN {X 0,Y 588.802,Z 602.448,A -85,B 0,C 180,E1 26154.096,E2 26154.096} C_VEL
LIN {X 0,Y 585.39,Z 601.896,A -85,B 0,C 180,E1 26153.531,E2 26153.531} C_VEL
LIN {X 0,Y 581.594,Z 600.135,A -85,B 0,C 180,E1 26153.074,E2 26153.074} C_VEL
LIN {X 0,Y 574.887,Z 595.079,A -85,B 0,C 180,E1 26152.311,E2 26152.311} C_VEL
LIN {X 0,Y 569.552,Z 588.731,A -85,B 0,C 180,E1 26151.532,E2 26151.532} C_VEL
LIN {X 0,Y 565.495,Z 581.037,A -85,B 0,C 180,E1 26150.73,E2 26150.73} C_VEL
LIN {X 0,Y 562.444,Z 570.884,A -85,B 0,C 180,E1 26149.812,E2 26149.812} C_VEL
LIN {X 0,Y 560.664,Z 557.719,A -85,B 0,C 180,E1 26148.759,E2 26148.759} C_VEL
LIN {X 0,Y 560.417,Z 537.65,A -85,B 0,C 180,E1 26147.312,E2 26147.312} C_VEL
LIN {X 0,Y 561.736,Z 500.064,A -85,B 0,C 180,E1 26144.605,E2 26144.605} C_VEL
LIN {X 0,Y 562.751,Z 468.813,A -85,B 0,C 180,E1 26142.26,E2 26142.26} C_VEL
LIN {X 0,Y 555.708,Z 454.339,A -85,B 0,C 180,E1 26140.37,E2 26140.37} C_VEL
LIN {X 0,Y 553.863,Z 450.482,A -85,B 0,C 180,E1 26139.856,E2 26139.856} C_VEL
LIN {X 0,Y 552.442,Z 447.352,A -85,B 0,C 180,E1 26139.44,E2 26139.44} C_VEL
LIN {X 0,Y 552.325,Z 446.69,A -85,B 0,C 180,E1 26139.353,E2 26139.353} C_VEL
LIN {X 0,Y 552.324,Z 446.687,A -85,B 0,C 180,E1 26136.039,E2 26136.039} C_VEL
LIN {X 0,Y 552.337,Z 446.682,A -85,B 0,C 180,E1 26132.769,E2 26132.769} C_VEL
LIN {X 0,Y 552.323,Z 446.687,A -85,B 0,C 180,E1 26129.456,E2 26129.456} C_VEL
LIN {X 0,Y 552.344,Z 446.685,A -85,B 0,C 180,E1 26126.096,E2 26126.096} C_VEL
LIN {X 0,Y 552.32,Z 446.687,A -85,B 0,C 180,E1 26122.68,E2 26122.68} C_VEL
LIN {X 0,Y 552.312,Z 446.688,A -85,B 0,C 180,E1 26119.347,E2 26119.347} C_VEL
LIN {X 0,Y 552.335,Z 446.686,A -85,B 0,C 180,E1 26116.079,E2 26116.079} C_VEL
LIN {X 0,Y 552.311,Z 446.689,A -85,B 0,C 180,E1 26112.759,E2 26112.759} C_VEL
LIN {X 0,Y 552.343,Z 446.683,A -85,B 0,C 180,E1 26109.376,E2 26109.376} C_VEL
LIN {X 0,Y 552.318,Z 446.686,A -85,B 0,C 180,E1 26106.027,E2 26106.027} C_VEL
LIN {X 0,Y 552.302,Z 446.688,A -85,B 0,C 180,E1 26102.698,E2 26102.698} C_VEL
LIN {X 0,Y 552.336,Z 446.684,A -85,B 0,C 180,E1 26099.481,E2 26099.481} C_VEL
LIN {X 0,Y 552.31,Z 446.687,A -85,B 0,C 180,E1 26096.159,E2 26096.159} C_VEL
LIN {X 0,Y 552.34,Z 446.677,A -85,B 0,C 180,E1 26092.72,E2 26092.72} C_VEL
LIN {X 0,Y 552.318,Z 446.685,A -85,B 0,C 180,E1 26089.359,E2 26089.359} C_VEL
LIN {X 0,Y 552.293,Z 446.686,A -85,B 0,C 180,E1 26085.96,E2 26085.96} C_VEL
LIN {X 0,Y 552.337,Z 446.68,A -85,B 0,C 180,E1 26082.838,E2 26082.838} C_VEL
LIN {X 0,Y 552.302,Z 446.687,A -85,B 0,C 180,E1 26079.439,E2 26079.439} C_VEL
LIN {X 0,Y 552.333,Z 446.683,A -85,B 0,C 180,E1 26076.078,E2 26076.078} C_VEL
LIN {X 0,Y 552.32,Z 446.683,A -85,B 0,C 180,E1 26072.728,E2 26072.728} C_VEL
LIN {X 0,Y 552.32,Z 446.682,A -85,B 0,C 180,E1 26072.689,E2 26072.689} C_VEL
LIN {X 0,Y 551.325,Z 446.809,A -85,B 0,C 180,E1 26071.89,E2 26071.89} C_VEL
LIN {X 0,Y 544.876,Z 447.612,A -85,B 0,C 180,E1 26069.646,E2 26069.646} C_VEL
LIN {X 0,Y 544.347,Z 447.673,A -85,B 0,C 180,E1 26069.061,E2 26069.061} C_VEL
LIN {X 0,Y 544.401,Z 447.669,A -85,B 0,C 180,E1 26065.738,E2 26065.738} C_VEL
LIN {X 0,Y 544.356,Z 447.675,A -85,B 0,C 180,E1 26062.424,E2 26062.424} C_VEL
LIN {X 0,Y 544.372,Z 447.671,A -85,B 0,C 180,E1 26059.015,E2 26059.015} C_VEL
LIN {X 0,Y 544.392,Z 447.673,A -85,B 0,C 180,E1 26055.739,E2 26055.739} C_VEL
LIN {X 0,Y 544.348,Z 447.68,A -85,B 0,C 180,E1 26052.384,E2 26052.384} C_VEL
LIN {X 0,Y 544.394,Z 447.673,A -85,B 0,C 180,E1 26049.022,E2 26049.022} C_VEL
LIN {X 0,Y 544.363,Z 447.679,A -85,B 0,C 180,E1 26045.723,E2 26045.723} C_VEL
LIN {X 0,Y 544.408,Z 447.733,A -85,B 0,C 180,E1 26045.114,E2 26045.114} C_VEL
LIN {X 0,Y 550.527,Z 464.953,A -85,B 0,C 180,E1 26043.263,E2 26043.263} C_VEL
LIN {X 0,Y 549.736,Z 495.405,A -85,B 0,C 180,E1 26040.854,E2 26040.854} C_VEL
LIN {X 0,Y 551.834,Z 507.434,A -85,B 0,C 180,E1 26040.546,E2 26040.546} C_VEL
LIN {X 0,Y 550.091,Z 754.667,A -85,B 0,C 180,E1 26037.015,E2 26037.015} C_VEL
LIN {X 0,Y 549.679,Z 775.938,A -85,B 0,C 180,E1 26036.528,E2 26036.528} C_VEL
LIN {X 0,Y 549.173,Z 796.436,A -85,B 0,C 180,E1 26035.851,E2 26035.851} C_VEL
LIN {X 0,Y 548.597,Z 815.785,A -85,B 0,C 180,E1 26035.013,E2 26035.013} C_VEL
LIN {X 0,Y 547.922,Z 834.907,A -85,B 0,C 180,E1 26033.978,E2 26033.978} C_VEL
LIN {X 0,Y 547.221,Z 853.697,A -85,B 0,C 180,E1 26032.733,E2 26032.733} C_VEL
LIN {X 0,Y 546.541,Z 871.033,A -85,B 0,C 180,E1 26031.349,E2 26031.349} C_VEL
LIN {X 0,Y 545.935,Z 886.65,A -85,B 0,C 180,E1 26029.877,E2 26029.877} C_VEL
LIN {X 0,Y 545.379,Z 901.347,A -85,B 0,C 180,E1 26028.256,E2 26028.256} C_VEL
LIN {X 0,Y 544.902,Z 915.517,A -85,B 0,C 180,E1 26026.414,E2 26026.414} C_VEL
LIN {X 0,Y 544.519,Z 928.135,A -85,B 0,C 180,E1 26024.461,E2 26024.461} C_VEL
LIN {X 0,Y 544.257,Z 939.13,A -85,B 0,C 180,E1 26022.412,E2 26022.412} C_VEL
LIN {X 0,Y 544.08,Z 948.09,A -85,B 0,C 180,E1 26020.375,E2 26020.375} C_VEL
LIN {X 0,Y 543.986,Z 955.567,A -85,B 0,C 180,E1 26018.242,E2 26018.242} C_VEL
LIN {X 0,Y 543.937,Z 961.356,A -85,B 0,C 180,E1 26016.032,E2 26016.032} C_VEL
LIN {X 0,Y 543.918,Z 965.174,A -85,B 0,C 180,E1 26013.899,E2 26013.899} C_VEL
LIN {X 0,Y 543.91,Z 967.346,A -85,B 0,C 180,E1 26011.79,E2 26011.79} C_VEL
LIN {X 0,Y 543.904,Z 967.949,A -85,B 0,C 180,E1 26009.683,E2 26009.683} C_VEL
LIN {X 0,Y 543.905,Z 966.992,A -85,B 0,C 180,E1 26007.576,E2 26007.576} C_VEL
LIN {X 0,Y 543.918,Z 964.201,A -85,B 0,C 180,E1 26005.36,E2 26005.36} C_VEL
LIN {X 0,Y 543.945,Z 959.843,A -85,B 0,C 180,E1 26003.243,E2 26003.243} C_VEL
LIN {X 0,Y 543.999,Z 953.772,A -85,B 0,C 180,E1 26001.118,E2 26001.118} C_VEL
LIN {X 0,Y 544.111,Z 945.829,A -85,B 0,C 180,E1 25998.982,E2 25998.982} C_VEL
LIN {X 0,Y 544.316,Z 936.366,A -85,B 0,C 180,E1 25996.941,E2 25996.941} C_VEL
LIN {X 0,Y 544.611,Z 925.147,A -85,B 0,C 180,E1 25994.949,E2 25994.949} C_VEL
LIN {X 0,Y 545.005,Z 912.272,A -85,B 0,C 180,E1 25993.04,E2 25993.04} C_VEL
LIN {X 0,Y 545.492,Z 898.281,A -85,B 0,C 180,E1 25991.29,E2 25991.29} C_VEL
LIN {X 0,Y 546.075,Z 882.747,A -85,B 0,C 180,E1 25989.641,E2 25989.641} C_VEL
LIN {X 0,Y 546.72,Z 866.319,A -85,B 0,C 180,E1 25988.164,E2 25988.164} C_VEL
LIN {X 0,Y 547.414,Z 848.577,A -85,B 0,C 180,E1 25986.82,E2 25986.82} C_VEL
LIN {X 0,Y 548.084,Z 830.037,A -85,B 0,C 180,E1 25985.651,E2 25985.651} C_VEL
LIN {X 0,Y 548.742,Z 810.476,A -85,B 0,C 180,E1 25984.647,E2 25984.647} C_VEL
LIN {X 0,Y 549.342,Z 790.679,A -85,B 0,C 180,E1 25983.846,E2 25983.846} C_VEL
LIN {X 0,Y 549.833,Z 770.158,A -85,B 0,C 180,E1 25983.225,E2 25983.225} C_VEL
LIN {X 0,Y 550.164,Z 748.964,A -85,B 0,C 180,E1 25982.796,E2 25982.796} C_VEL
LIN {X 0,Y 551.714,Z 511.033,A -85,B 0,C 180,E1 25979.41,E2 25979.41} C_VEL
LIN {X 0,Y 548.076,Z 497.358,A -85,B 0,C 180,E1 25978.962,E2 25978.962} C_VEL
LIN {X 0,Y 548.891,Z 472.827,A -85,B 0,C 180,E1 25975.997,E2 25975.997} C_VEL
LIN {X 0,Y 549.11,Z 463.292,A -85,B 0,C 180,E1 25974.843,E2 25974.843} C_VEL
LIN {X 0,Y 544.385,Z 447.677,A -85,B 0,C 180,E1 25972.559,E2 25972.559} C_VEL
LIN {X 0,Y 544.405,Z 447.677,A -85,B 0,C 180,E1 25969.168,E2 25969.168} C_VEL
LIN {X 0,Y 544.371,Z 447.672,A -85,B 0,C 180,E1 25965.883,E2 25965.883} C_VEL
LIN {X 0,Y 544.4,Z 447.668,A -85,B 0,C 180,E1 25962.523,E2 25962.523} C_VEL
LIN {X 0,Y 544.399,Z 447.676,A -85,B 0,C 180,E1 25959.048,E2 25959.048} C_VEL
LIN {X 0,Y 544.39,Z 447.676,A -85,B 0,C 180,E1 25955.607,E2 25955.607} C_VEL
LIN {X 0,Y 544.399,Z 447.675,A -85,B 0,C 180,E1 25952.183,E2 25952.183} C_VEL
LIN {X 0,Y 544.44,Z 447.909,A -85,B 0,C 180,E1 25949.935,E2 25949.935} C_VEL
LIN {X 0,Y 549.751,Z 464.264,A -85,B 0,C 180,E1 25947.92,E2 25947.92} C_VEL
LIN {X 0,Y 548.955,Z 495.804,A -85,B 0,C 180,E1 25944.882,E2 25944.882} C_VEL
LIN {X 0,Y 547.997,Z 529.569,A -85,B 0,C 180,E1 25941.683,E2 25941.683} C_VEL
LIN {X 0,Y 547.031,Z 565.522,A -85,B 0,C 180,E1 25938.324,E2 25938.324} C_VEL
LIN {X 0,Y 546.225,Z 600.658,A -85,B 0,C 180,E1 25935.066,E2 25935.066} C_VEL
LIN {X 0,Y 546.198,Z 605.152,A -85,B 0,C 180,E1 25934.68,E2 25934.68} C_VEL
LIN {X 0,Y 546.749,Z 611.786,A -85,B 0,C 180,E1 25934.557,E2 25934.557} C_VEL
LIN {X 0,Y 546.046,Z 743.776,A -85,B 0,C 180,E1 25932.717,E2 25932.717} C_VEL
LIN {X 0,Y 545.908,Z 759.51,A -85,B 0,C 180,E1 25932.344,E2 25932.344} C_VEL
LIN {X 0,Y 545.698,Z 774.538,A -85,B 0,C 180,E1 25931.789,E2 25931.789} C_VEL
LIN {X 0,Y 545.44,Z 787.418,A -85,B 0,C 180,E1 25931.151,E2 25931.151} C_VEL
LIN {X 0,Y 545.178,Z 800.17,A -85,B 0,C 180,E1 25930.354,E2 25930.354} C_VEL
LIN {X 0,Y 544.85,Z 814.193,A -85,B 0,C 180,E1 25929.24,E2 25929.24} C_VEL
LIN {X 0,Y 544.592,Z 824.342,A -85,B 0,C 180,E1 25928.234,E2 25928.234} C_VEL
LIN {X 0,Y 544.376,Z 833.252,A -85,B 0,C 180,E1 25927.175,E2 25927.175} C_VEL
LIN {X 0,Y 544.179,Z 842.809,A -85,B 0,C 180,E1 25925.8,E2 25925.8} C_VEL
LIN {X 0,Y 544.033,Z 850.765,A -85,B 0,C 180,E1 25924.322,E2 25924.322} C_VEL
LIN {X 0,Y 543.969,Z 856.354,A -85,B 0,C 180,E1 25923.056,E2 25923.056} C_VEL
LIN {X 0,Y 543.935,Z 861.073,A -85,B 0,C 180,E1 25921.686,E2 25921.686} C_VEL
LIN {X 0,Y 543.921,Z 865.198,A -85,B 0,C 180,E1 25920,E2 25920} C_VEL
LIN {X 0,Y 543.913,Z 867.361,A -85,B 0,C 180,E1 25918.315,E2 25918.315} C_VEL
LIN {X 0,Y 543.915,Z 867.912,A -85,B 0,C 180,E1 25916.944,E2 25916.944} C_VEL
LIN {X 0,Y 543.915,Z 867.265,A -85,B 0,C 180,E1 25915.466,E2 25915.466} C_VEL
LIN {X 0,Y 543.92,Z 864.693,A -85,B 0,C 180,E1 25913.668,E2 25913.668} C_VEL
LIN {X 0,Y 543.939,Z 860.943,A -85,B 0,C 180,E1 25912.182,E2 25912.182} C_VEL
LIN {X 0,Y 543.971,Z 856.552,A -85,B 0,C 180,E1 25910.905,E2 25910.905} C_VEL
LIN {X 0,Y 544.062,Z 849.51,A -85,B 0,C 180,E1 25909.303,E2 25909.303} C_VEL
LIN {X 0,Y 544.229,Z 840.898,A -85,B 0,C 180,E1 25907.796,E2 25907.796} C_VEL
LIN {X 0,Y 544.427,Z 832.598,A -85,B 0,C 180,E1 25906.62,E2 25906.62} C_VEL
LIN {X 0,Y 544.716,Z 821.972,A -85,B 0,C 180,E1 25905.381,E2 25905.381} C_VEL
LIN {X 0,Y 545.048,Z 809.213,A -85,B 0,C 180,E1 25904.207,E2 25904.207} C_VEL
LIN {X 0,Y 545.329,Z 797.297,A -85,B 0,C 180,E1 25903.325,E2 25903.325} C_VEL
LIN {X 0,Y 545.613,Z 783.513,A -85,B 0,C 180,E1 25902.51,E2 25902.51} C_VEL
LIN {X 0,Y 545.855,Z 767.874,A -85,B 0,C 180,E1 25901.829,E2 25901.829} C_VEL
LIN {X 0,Y 546.006,Z 752.98,A -85,B 0,C 180,E1 25901.373,E2 25901.373} C_VEL
LIN {X 0,Y 546.137,Z 732.743,A -85,B 0,C 180,E1 25901.014,E2 25901.014} C_VEL
LIN {X 0,Y 547.046,Z 615.191,A -85,B 0,C 180,E1 25899.313,E2 25899.313} C_VEL
LIN {X 0,Y 547.088,Z 608.933,A -85,B 0,C 180,E1 25899.206,E2 25899.206} C_VEL
LIN {X 0,Y 548.528,Z 582.378,A -85,B 0,C 180,E1 25896.586,E2 25896.586} C_VEL
LIN {X 0,Y 550.892,Z 547.007,A -85,B 0,C 180,E1 25892.958,E2 25892.958} C_VEL
LIN {X 0,Y 554.131,Z 514.34,A -85,B 0,C 180,E1 25889.414,E2 25889.414} C_VEL
LIN {X 0,Y 557.121,Z 492.514,A -85,B 0,C 180,E1 25886.874,E2 25886.874} C_VEL
LIN {X 0,Y 559.104,Z 478.188,A -85,B 0,C 180,E1 25884.967,E2 25884.967} C_VEL
LIN {X 0,Y 557.313,Z 473.402,A -85,B 0,C 180,E1 25883.663,E2 25883.663} C_VEL
LIN {X 0,Y 556.628,Z 471.357,A -85,B 0,C 180,E1 25883.005,E2 25883.005} C_VEL
LIN {X 0,Y 555.687,Z 468.23,A -85,B 0,C 180,E1 25881.628,E2 25881.628} C_VEL
LIN {X 0,Y 555.182,Z 467.417,A -85,B 0,C 180,E1 25880.258,E2 25880.258} C_VEL
LIN {X 0,Y 555.842,Z 468.204,A -85,B 0,C 180,E1 25879.07,E2 25879.07} C_VEL
LIN {X 0,Y 556.475,Z 469.418,A -85,B 0,C 180,E1 25878.47,E2 25878.47} C_VEL
LIN {X 0,Y 557.543,Z 472.562,A -85,B 0,C 180,E1 25877.601,E2 25877.601} C_VEL
LIN {X 0,Y 557.54,Z 473.827,A -85,B 0,C 180,E1 25877.407,E2 25877.407} C_VEL
LIN {X 0,Y 554.414,Z 489.475,A -85,B 0,C 180,E1 25876.02,E2 25876.02} C_VEL
LIN {X 0,Y 551.722,Z 512.34,A -85,B 0,C 180,E1 25874.245,E2 25874.245} C_VEL
LIN {X 0,Y 550.085,Z 542.348,A -85,B 0,C 180,E1 25872.123,E2 25872.123} C_VEL
LIN {X 0,Y 551.129,Z 561.173,A -85,B 0,C 180,E1 25870.777,E2 25870.777} C_VEL
LIN {X 0,Y 553.711,Z 574.111,A -85,B 0,C 180,E1 25869.795,E2 25869.795} C_VEL
LIN {X 0,Y 557.736,Z 584.936,A -85,B 0,C 180,E1 25868.919,E2 25868.919} C_VEL
LIN {X 0,Y 563.124,Z 593.817,A -85,B 0,C 180,E1 25868.134,E2 25868.134} C_VEL
LIN {X 0,Y 570.052,Z 601.346,A -85,B 0,C 180,E1 25867.387,E2 25867.387} C_VEL
LIN {X 0,Y 577.634,Z 606.928,A -85,B 0,C 180,E1 25866.733,E2 25866.733} C_VEL
LIN {X 0,Y 581.829,Z 608.869,A -85,B 0,C 180,E1 25866.297,E2 25866.297} C_VEL
LIN {X 0,Y 585.445,Z 609.617,A -85,B 0,C 180,E1 25865.784,E2 25865.784} C_VEL
LIN {X 0,Y 588.276,Z 609.08,A -85,B 0,C 180,E1 25865.183,E2 25865.183} C_VEL
LIN {X 0,Y 589.688,Z 607.476,A -85,B 0,C 180,E1 25864.613,E2 25864.613} C_VEL
LIN {X 0,Y 589.793,Z 604.649,A -85,B 0,C 180,E1 25864.018,E2 25864.018} C_VEL
LIN {X 0,Y 588.421,Z 600.975,A -85,B 0,C 180,E1 25863.493,E2 25863.493} C_VEL
LIN {X 0,Y 584.487,Z 594.215,A -85,B 0,C 180,E1 25862.854,E2 25862.854} C_VEL
LIN {X 0,Y 580.454,Z 585.204,A -85,B 0,C 180,E1 25862.232,E2 25862.232} C_VEL
LIN {X 0,Y 577.21,Z 574.924,A -85,B 0,C 180,E1 25861.718,E2 25861.718} C_VEL
LIN {X 0,Y 574.792,Z 563.411,A -85,B 0,C 180,E1 25861.326,E2 25861.326} C_VEL
LIN {X 0,Y 574.273,Z 560.516,A -85,B 0,C 180,E1 25861.241,E2 25861.241} C_VEL
LIN {X 0,Y 573.328,Z 565.007,A -85,B 0,C 180,E1 25861.085,E2 25861.085} C_VEL
LIN {X 0,Y 569.01,Z 624.463,A -85,B 0,C 180,E1 25860.356,E2 25860.356} C_VEL
LIN {X 0,Y 565.287,Z 665.84,A -85,B 0,C 180,E1 25859.705,E2 25859.705} C_VEL
LIN {X 0,Y 562.947,Z 684.596,A -85,B 0,C 180,E1 25859.289,E2 25859.289} C_VEL
LIN {X 0,Y 561.409,Z 692.114,A -85,B 0,C 180,E1 25859.02,E2 25859.02} C_VEL
LIN {X 0,Y 558.808,Z 710.834,A -85,B 0,C 180,E1 25858.838,E2 25858.838} C_VEL
LIN {X 0,Y 555.161,Z 726.753,A -85,B 0,C 180,E1 25858.581,E2 25858.581} C_VEL
LIN {X 0,Y 551.986,Z 738.676,A -85,B 0,C 180,E1 25858.215,E2 25858.215} C_VEL
LIN {X 0,Y 550.522,Z 745.008,A -85,B 0,C 180,E1 25857.923,E2 25857.923} C_VEL
LIN {X 0,Y 550.063,Z 807.063,A -85,B 0,C 180,E1 25857.018,E2 25857.018} C_VEL
LIN {X 0,Y 549.642,Z 828.414,A -85,B 0,C 180,E1 25856.504,E2 25856.504} C_VEL
LIN {X 0,Y 549.126,Z 848.341,A -85,B 0,C 180,E1 25855.826,E2 25855.826} C_VEL
LIN {X 0,Y 548.527,Z 867.767,A -85,B 0,C 180,E1 25854.96,E2 25854.96} C_VEL
LIN {X 0,Y 547.846,Z 887.164,A -85,B 0,C 180,E1 25853.885,E2 25853.885} C_VEL
LIN {X 0,Y 547.153,Z 905.299,A -85,B 0,C 180,E1 25852.657,E2 25852.657} C_VEL
LIN {X 0,Y 546.466,Z 922.788,A -85,B 0,C 180,E1 25851.241,E2 25851.241} C_VEL
LIN {X 0,Y 545.801,Z 939.867,A -85,B 0,C 180,E1 25849.588,E2 25849.588} C_VEL
LIN {X 0,Y 545.308,Z 953.404,A -85,B 0,C 180,E1 25848.052,E2 25848.052} C_VEL
LIN {X 0,Y 544.841,Z 967.344,A -85,B 0,C 180,E1 25846.198,E2 25846.198} C_VEL
LIN {X 0,Y 544.497,Z 979.016,A -85,B 0,C 180,E1 25844.354,E2 25844.354} C_VEL
LIN {X 0,Y 544.239,Z 989.859,A -85,B 0,C 180,E1 25842.305,E2 25842.305} C_VEL
LIN {X 0,Y 544.069,Z 998.683,A -85,B 0,C 180,E1 25840.269,E2 25840.269} C_VEL
LIN {X 0,Y 543.978,Z 1005.972,A -85,B 0,C 180,E1 25838.137,E2 25838.137} C_VEL
LIN {X 0,Y 543.937,Z 1011.237,A -85,B 0,C 180,E1 25836.121,E2 25836.121} C_VEL
LIN {X 0,Y 543.918,Z 1015.258,A -85,B 0,C 180,E1 25833.901,E2 25833.901} C_VEL
LIN {X 0,Y 543.909,Z 1017.39,A -85,B 0,C 180,E1 25831.791,E2 25831.791} C_VEL
LIN {X 0,Y 543.9,Z 1017.918,A -85,B 0,C 180,E1 25829.579,E2 25829.579} C_VEL
LIN {X 0,Y 543.908,Z 1016.838,A -85,B 0,C 180,E1 25827.472,E2 25827.472} C_VEL
LIN {X 0,Y 543.92,Z 1013.95,A -85,B 0,C 180,E1 25825.256,E2 25825.256} C_VEL
LIN {X 0,Y 543.946,Z 1009.724,A -85,B 0,C 180,E1 25823.245,E2 25823.245} C_VEL
LIN {X 0,Y 543.998,Z 1003.646,A -85,B 0,C 180,E1 25821.119,E2 25821.119} C_VEL
LIN {X 0,Y 544.107,Z 996.096,A -85,B 0,C 180,E1 25819.09,E2 25819.09} C_VEL
LIN {X 0,Y 544.311,Z 986.704,A -85,B 0,C 180,E1 25817.05,E2 25817.05} C_VEL
LIN {X 0,Y 544.563,Z 976.442,A -85,B 0,C 180,E1 25815.214,E2 25815.214} C_VEL
LIN {X 0,Y 544.965,Z 963.529,A -85,B 0,C 180,E1 25813.259,E2 25813.259} C_VEL
LIN {X 0,Y 545.432,Z 949.742,A -85,B 0,C 180,E1 25811.511,E2 25811.511} C_VEL
LIN {X 0,Y 546.05,Z 933.421,A -85,B 0,C 180,E1 25809.753,E2 25809.753} C_VEL
LIN {X 0,Y 546.689,Z 917.373,A -85,B 0,C 180,E1 25808.294,E2 25808.294} C_VEL
LIN {X 0,Y 547.413,Z 898.806,A -85,B 0,C 180,E1 25806.878,E2 25806.878} C_VEL
LIN {X 0,Y 548.096,Z 880.009,A -85,B 0,C 180,E1 25805.691,E2 25805.691} C_VEL
LIN {X 0,Y 548.739,Z 860.811,A -85,B 0,C 180,E1 25804.705,E2 25804.705} C_VEL
LIN {X 0,Y 549.342,Z 840.852,A -85,B 0,C 180,E1 25803.896,E2 25803.896} C_VEL
LIN {X 0,Y 549.824,Z 820.306,A -85,B 0,C 180,E1 25803.274,E2 25803.274} C_VEL
LIN {X 0,Y 550.152,Z 799.046,A -85,B 0,C 180,E1 25802.844,E2 25802.844} C_VEL
LIN {X 0,Y 550.604,Z 743.985,A -85,B 0,C 180,E1 25802.048,E2 25802.048} C_VEL
LIN {X 0,Y 552.919,Z 735.193,A -85,B 0,C 180,E1 25801.654,E2 25801.654} C_VEL
LIN {X 0,Y 556.414,Z 721.766,A -85,B 0,C 180,E1 25801.318,E2 25801.318} C_VEL
LIN {X 0,Y 559.9,Z 704.574,A -85,B 0,C 180,E1 25801.097,E2 25801.097} C_VEL
LIN {X 0,Y 561.618,Z 690.721,A -85,B 0,C 180,E1 25800.947,E2 25800.947} C_VEL
LIN {X 0,Y 563.117,Z 683.569,A -85,B 0,C 180,E1 25800.682,E2 25800.682} C_VEL
LIN {X 0,Y 565.608,Z 662.723,A -85,B 0,C 180,E1 25800.238,E2 25800.238} C_VEL
LIN {X 0,Y 569.47,Z 618.687,A -85,B 0,C 180,E1 25799.565,E2 25799.565} C_VEL
LIN {X 0,Y 573.555,Z 563.489,A -85,B 0,C 180,E1 25798.878,E2 25798.878} C_VEL
LIN {X 0,Y 574.348,Z 560.529,A -85,B 0,C 180,E1 25798.747,E2 25798.747} C_VEL
LIN {X 0,Y 576.613,Z 572.547,A -85,B 0,C 180,E1 25798.378,E2 25798.378} C_VEL
LIN {X 0,Y 579.715,Z 583.204,A -85,B 0,C 180,E1 25797.883,E2 25797.883} C_VEL
LIN {X 0,Y 583.668,Z 592.617,A -85,B 0,C 180,E1 25797.27,E2 25797.27} C_VEL
LIN {X 0,Y 588.107,Z 600.385,A -85,B 0,C 180,E1 25796.576,E2 25796.576} C_VEL
LIN {X 0,Y 589.684,Z 604.147,A -85,B 0,C 180,E1 25796.064,E2 25796.064} C_VEL
LIN {X 0,Y 589.795,Z 607.138,A -85,B 0,C 180,E1 25795.477,E2 25795.477} C_VEL
LIN {X 0,Y 588.709,Z 608.795,A -85,B 0,C 180,E1 25794.947,E2 25794.947} C_VEL
LIN {X 0,Y 586.497,Z 609.6,A -85,B 0,C 180,E1 25794.408,E2 25794.408} C_VEL
LIN {X 0,Y 582.916,Z 609.198,A -85,B 0,C 180,E1 25793.84,E2 25793.84} C_VEL
LIN {X 0,Y 578.375,Z 607.332,A -85,B 0,C 180,E1 25793.334,E2 25793.334} C_VEL
LIN {X 0,Y 570.822,Z 602.182,A -85,B 0,C 180,E1 25792.512,E2 25792.512} C_VEL
LIN {X 0,Y 564.7,Z 595.626,A -85,B 0,C 180,E1 25791.663,E2 25791.663} C_VEL
LIN {X 0,Y 559.764,Z 587.212,A -85,B 0,C 180,E1 25790.743,E2 25790.743} C_VEL
LIN {X 0,Y 556.364,Z 577.176,A -85,B 0,C 180,E1 25789.798,E2 25789.798} C_VEL
LIN {X 0,Y 554.269,Z 565.073,A -85,B 0,C 180,E1 25788.784,E2 25788.784} C_VEL
LIN {X 0,Y 553.555,Z 547.186,A -85,B 0,C 180,E1 25787.442,E2 25787.442} C_VEL
LIN {X 0,Y 555.169,Z 504.683,A -85,B 0,C 180,E1 25784.358,E2 25784.358} C_VEL
LIN {X 0,Y 556.381,Z 472.842,A -85,B 0,C 180,E1 25781.952,E2 25781.952} C_VEL
LIN {X 0,Y 547.863,Z 455.46,A -85,B 0,C 180,E1 25779.633,E2 25779.633} C_VEL
LIN {X 0,Y 545.812,Z 451.354,A -85,B 0,C 180,E1 25779.062,E2 25779.062} C_VEL
LIN {X 0,Y 544.416,Z 447.932,A -85,B 0,C 180,E1 25778.615,E2 25778.615} C_VEL
LIN {X 0,Y 544.357,Z 447.677,A -85,B 0,C 180,E1 25777.443,E2 25777.443} C_VEL
LIN {X 0,Y 544.4,Z 447.671,A -85,B 0,C 180,E1 25774.067,E2 25774.067} C_VEL
LIN {X 0,Y 544.373,Z 447.675,A -85,B 0,C 180,E1 25770.704,E2 25770.704} C_VEL
LIN {X 0,Y 544.355,Z 447.677,A -85,B 0,C 180,E1 25767.217,E2 25767.217} C_VEL
LIN {X 0,Y 544.4,Z 447.671,A -85,B 0,C 180,E1 25763.947,E2 25763.947} C_VEL
LIN {X 0,Y 544.351,Z 447.677,A -85,B 0,C 180,E1 25760.65,E2 25760.65} C_VEL
LIN {X 0,Y 544.381,Z 447.674,A -85,B 0,C 180,E1 25757.2,E2 25757.2} C_VEL
LIN {X 0,Y 544.377,Z 447.674,A -85,B 0,C 180,E1 25753.922,E2 25753.922} C_VEL
LIN {X 0,Y 544.35,Z 447.677,A -85,B 0,C 180,E1 25750.477,E2 25750.477} C_VEL
LIN {X 0,Y 544.403,Z 447.67,A -85,B 0,C 180,E1 25747.174,E2 25747.174} C_VEL
LIN {X 0,Y 544.348,Z 447.677,A -85,B 0,C 180,E1 25743.897,E2 25743.897} C_VEL
LIN {X 0,Y 544.376,Z 447.673,A -85,B 0,C 180,E1 25740.421,E2 25740.421} C_VEL
LIN {X 0,Y 544.386,Z 447.672,A -85,B 0,C 180,E1 25737.157,E2 25737.157} C_VEL
LIN {X 0,Y 544.351,Z 447.676,A -85,B 0,C 180,E1 25733.778,E2 25733.778} C_VEL
LIN {X 0,Y 544.396,Z 447.67,A -85,B 0,C 180,E1 25730.379,E2 25730.379} C_VEL
LIN {X 0,Y 544.355,Z 447.671,A -85,B 0,C 180,E1 25727.159,E2 25727.159} C_VEL
LIN {X 0,Y 544.374,Z 447.674,A -85,B 0,C 180,E1 25723.789,E2 25723.789} C_VEL
LIN {X 0,Y 544.4,Z 447.67,A -85,B 0,C 180,E1 25720.421,E2 25720.421} C_VEL
LIN {X 0,Y 544.356,Z 447.671,A -85,B 0,C 180,E1 25717.083,E2 25717.083} C_VEL
LIN {X 0,Y 544.393,Z 447.672,A -85,B 0,C 180,E1 25713.673,E2 25713.673} C_VEL
LIN {X 0,Y 544.368,Z 447.677,A -85,B 0,C 180,E1 25710.391,E2 25710.391} C_VEL
LIN {X 0,Y 544.347,Z 447.673,A -85,B 0,C 180,E1 25709.061,E2 25709.061} C_VEL
LIN {X 0,Y 543.372,Z 447.802,A -85,B 0,C 180,E1 25708.25,E2 25708.25} C_VEL
LIN {X 0,Y 536.89,Z 448.606,A -85,B 0,C 180,E1 25705.913,E2 25705.913} C_VEL
LIN {X 0,Y 536.454,Z 448.66,A -85,B 0,C 180,E1 25705.379,E2 25705.379} C_VEL
LIN {X 0,Y 536.434,Z 448.663,A -85,B 0,C 180,E1 25702.038,E2 25702.038} C_VEL
LIN {X 0,Y 536.439,Z 448.661,A -85,B 0,C 180,E1 25698.689,E2 25698.689} C_VEL
LIN {X 0,Y 536.466,Z 448.664,A -85,B 0,C 180,E1 25695.243,E2 25695.243} C_VEL
LIN {X 0,Y 536.45,Z 448.664,A -85,B 0,C 180,E1 25691.795,E2 25691.795} C_VEL
LIN {X 0,Y 536.461,Z 448.665,A -85,B 0,C 180,E1 25688.363,E2 25688.363} C_VEL
LIN {X 0,Y 536.436,Z 448.729,A -85,B 0,C 180,E1 25685.62,E2 25685.62} C_VEL
LIN {X 0,Y 543.4,Z 468.007,A -85,B 0,C 180,E1 25683.504,E2 25683.504} C_VEL
LIN {X 0,Y 542.601,Z 495.482,A -85,B 0,C 180,E1 25681.306,E2 25681.306} C_VEL
LIN {X 0,Y 544.938,Z 508.865,A -85,B 0,C 180,E1 25680.954,E2 25680.954} C_VEL
LIN {X 0,Y 542.956,Z 755.078,A -85,B 0,C 180,E1 25677.392,E2 25677.392} C_VEL
LIN {X 0,Y 542.489,Z 776.336,A -85,B 0,C 180,E1 25676.896,E2 25676.896} C_VEL
LIN {X 0,Y 541.932,Z 796.446,A -85,B 0,C 180,E1 25676.223,E2 25676.223} C_VEL
LIN {X 0,Y 541.276,Z 815.805,A -85,B 0,C 180,E1 25675.375,E2 25675.375} C_VEL
LIN {X 0,Y 540.53,Z 834.392,A -85,B 0,C 180,E1 25674.361,E2 25674.361} C_VEL
LIN {X 0,Y 539.752,Z 852.912,A -85,B 0,C 180,E1 25673.123,E2 25673.123} C_VEL
LIN {X 0,Y 538.998,Z 869.727,A -85,B 0,C 180,E1 25671.777,E2 25671.777} C_VEL
LIN {X 0,Y 538.282,Z 885.658,A -85,B 0,C 180,E1 25670.275,E2 25670.275} C_VEL
LIN {X 0,Y 537.613,Z 901.236,A -85,B 0,C 180,E1 25668.543,E2 25668.543} C_VEL
LIN {X 0,Y 537.058,Z 915.519,A -85,B 0,C 180,E1 25666.66,E2 25666.66} C_VEL
LIN {X 0,Y 536.619,Z 928.141,A -85,B 0,C 180,E1 25664.678,E2 25664.678} C_VEL
LIN {X 0,Y 536.314,Z 939.135,A -85,B 0,C 180,E1 25662.598,E2 25662.598} C_VEL
LIN {X 0,Y 536.112,Z 948.094,A -85,B 0,C 180,E1 25660.531,E2 25660.531} C_VEL
LIN {X 0,Y 536.001,Z 955.569,A -85,B 0,C 180,E1 25658.366,E2 25658.366} C_VEL
LIN {X 0,Y 535.941,Z 961.149,A -85,B 0,C 180,E1 25656.211,E2 25656.211} C_VEL
LIN {X 0,Y 535.92,Z 965.017,A -85,B 0,C 180,E1 25654.065,E2 25654.065} C_VEL
LIN {X 0,Y 535.911,Z 967.346,A -85,B 0,C 180,E1 25651.817,E2 25651.817} C_VEL
LIN {X 0,Y 535.904,Z 967.949,A -85,B 0,C 180,E1 25649.679,E2 25649.679} C_VEL
LIN {X 0,Y 535.905,Z 966.992,A -85,B 0,C 180,E1 25647.54,E2 25647.54} C_VEL
LIN {X 0,Y 535.919,Z 964.358,A -85,B 0,C 180,E1 25645.398,E2 25645.398} C_VEL
LIN {X 0,Y 535.948,Z 960.095,A -85,B 0,C 180,E1 25643.25,E2 25643.25} C_VEL
LIN {X 0,Y 536.009,Z 954.118,A -85,B 0,C 180,E1 25641.093,E2 25641.093} C_VEL
LIN {X 0,Y 536.13,Z 946.732,A -85,B 0,C 180,E1 25639.033,E2 25639.033} C_VEL
LIN {X 0,Y 536.357,Z 937.482,A -85,B 0,C 180,E1 25636.963,E2 25636.963} C_VEL
LIN {X 0,Y 536.668,Z 926.736,A -85,B 0,C 180,E1 25634.991,E2 25634.991} C_VEL
LIN {X 0,Y 537.09,Z 914.569,A -85,B 0,C 180,E1 25633.113,E2 25633.113} C_VEL
LIN {X 0,Y 537.66,Z 900.131,A -85,B 0,C 180,E1 25631.232,E2 25631.232} C_VEL
LIN {X 0,Y 538.333,Z 884.393,A -85,B 0,C 180,E1 25629.506,E2 25629.506} C_VEL
LIN {X 0,Y 539.091,Z 867.462,A -85,B 0,C 180,E1 25627.939,E2 25627.939} C_VEL
LIN {X 0,Y 539.9,Z 849.36,A -85,B 0,C 180,E1 25626.536,E2 25626.536} C_VEL
LIN {X 0,Y 540.661,Z 831.002,A -85,B 0,C 180,E1 25625.353,E2 25625.353} C_VEL
LIN {X 0,Y 541.394,Z 812.117,A -85,B 0,C 180,E1 25624.356,E2 25624.356} C_VEL
LIN {X 0,Y 542.088,Z 792.053,A -85,B 0,C 180,E1 25623.519,E2 25623.519} C_VEL
LIN {X 0,Y 542.644,Z 771.22,A -85,B 0,C 180,E1 25622.871,E2 25622.871} C_VEL
LIN {X 0,Y 543.03,Z 750.119,A -85,B 0,C 180,E1 25622.428,E2 25622.428} C_VEL
LIN {X 0,Y 544.834,Z 512.822,A -85,B 0,C 180,E1 25619.009,E2 25619.009} C_VEL
LIN {X 0,Y 540.736,Z 497.591,A -85,B 0,C 180,E1 25618.502,E2 25618.502} C_VEL
LIN {X 0,Y 541.619,Z 473.828,A -85,B 0,C 180,E1 25615.604,E2 25615.604} C_VEL
LIN {X 0,Y 541.775,Z 466.111,A -85,B 0,C 180,E1 25614.659,E2 25614.659} C_VEL
LIN {X 0,Y 536.422,Z 448.669,A -85,B 0,C 180,E1 25612.04,E2 25612.04} C_VEL
LIN {X 0,Y 536.467,Z 448.661,A -85,B 0,C 180,E1 25608.686,E2 25608.686} C_VEL
LIN {X 0,Y 536.461,Z 448.666,A -85,B 0,C 180,E1 25605.209,E2 25605.209} C_VEL
LIN {X 0,Y 536.44,Z 448.661,A -85,B 0,C 180,E1 25601.793,E2 25601.793} C_VEL
LIN {X 0,Y 536.458,Z 448.66,A -85,B 0,C 180,E1 25598.481,E2 25598.481} C_VEL
LIN {X 0,Y 536.458,Z 448.667,A -85,B 0,C 180,E1 25595.034,E2 25595.034} C_VEL
LIN {X 0,Y 536.457,Z 448.669,A -85,B 0,C 180,E1 25591.583,E2 25591.583} C_VEL
LIN {X 0,Y 536.461,Z 448.79,A -85,B 0,C 180,E1 25590.444,E2 25590.444} C_VEL
LIN {X 0,Y 542.548,Z 467.035,A -85,B 0,C 180,E1 25588.15,E2 25588.15} C_VEL
LIN {X 0,Y 541.641,Z 498.801,A -85,B 0,C 180,E1 25585.066,E2 25585.066} C_VEL
LIN {X 0,Y 540.602,Z 532.965,A -85,B 0,C 180,E1 25581.802,E2 25581.802} C_VEL
LIN {X 0,Y 539.531,Z 569.019,A -85,B 0,C 180,E1 25578.405,E2 25578.405} C_VEL
LIN {X 0,Y 538.642,Z 604.81,A -85,B 0,C 180,E1 25575.063,E2 25575.063} C_VEL
LIN {X 0,Y 538.752,Z 606.475,A -85,B 0,C 180,E1 25574.961,E2 25574.961} C_VEL
LIN {X 0,Y 539.257,Z 612.764,A -85,B 0,C 180,E1 25574.843,E2 25574.843} C_VEL
LIN {X 0,Y 538.371,Z 745.875,A -85,B 0,C 180,E1 25572.925,E2 25572.925} C_VEL
LIN {X 0,Y 538.208,Z 762.376,A -85,B 0,C 180,E1 25572.503,E2 25572.503} C_VEL
LIN {X 0,Y 537.971,Z 777.617,A -85,B 0,C 180,E1 25571.906,E2 25571.906} C_VEL
LIN {X 0,Y 537.678,Z 791.996,A -85,B 0,C 180,E1 25571.151,E2 25571.151} C_VEL
LIN {X 0,Y 537.312,Z 806.723,A -85,B 0,C 180,E1 25570.133,E2 25570.133} C_VEL
LIN {X 0,Y 536.999,Z 818.504,A -85,B 0,C 180,E1 25569.106,E2 25569.106} C_VEL
LIN {X 0,Y 536.677,Z 830.494,A -85,B 0,C 180,E1 25567.817,E2 25567.817} C_VEL
LIN {X 0,Y 536.424,Z 840.001,A -85,B 0,C 180,E1 25566.529,E2 25566.529} C_VEL
LIN {X 0,Y 536.25,Z 847.757,A -85,B 0,C 180,E1 25565.242,E2 25565.242} C_VEL
LIN {X 0,Y 536.111,Z 855.019,A -85,B 0,C 180,E1 25563.743,E2 25563.743} C_VEL
LIN {X 0,Y 536.013,Z 860.797,A -85,B 0,C 180,E1 25562.138,E2 25562.138} C_VEL
LIN {X 0,Y 535.971,Z 864.663,A -85,B 0,C 180,E1 25560.642,E2 25560.642} C_VEL
LIN {X 0,Y 535.949,Z 867.361,A -85,B 0,C 180,E1 25559.038,E2 25559.038} C_VEL
LIN {X 0,Y 535.942,Z 868.562,A -85,B 0,C 180,E1 25557.22,E2 25557.22} C_VEL
LIN {X 0,Y 535.944,Z 868.078,A -85,B 0,C 180,E1 25555.613,E2 25555.613} C_VEL
LIN {X 0,Y 535.965,Z 866.042,A -85,B 0,C 180,E1 25553.896,E2 25553.896} C_VEL
LIN {X 0,Y 536.022,Z 862.127,A -85,B 0,C 180,E1 25552.174,E2 25552.174} C_VEL
LIN {X 0,Y 536.113,Z 857.182,A -85,B 0,C 180,E1 25550.662,E2 25550.662} C_VEL
LIN {X 0,Y 536.263,Z 850.099,A -85,B 0,C 180,E1 25549.037,E2 25549.037} C_VEL
LIN {X 0,Y 536.464,Z 841.837,A -85,B 0,C 180,E1 25547.591,E2 25547.591} C_VEL
LIN {X 0,Y 536.716,Z 832.826,A -85,B 0,C 180,E1 25546.315,E2 25546.315} C_VEL
LIN {X 0,Y 537.079,Z 820.768,A -85,B 0,C 180,E1 25544.948,E2 25544.948} C_VEL
LIN {X 0,Y 537.42,Z 808.536,A -85,B 0,C 180,E1 25543.851,E2 25543.851} C_VEL
LIN {X 0,Y 537.755,Z 794.97,A -85,B 0,C 180,E1 25542.882,E2 25542.882} C_VEL
LIN {X 0,Y 538.055,Z 780.238,A -85,B 0,C 180,E1 25542.073,E2 25542.073} C_VEL
LIN {X 0,Y 538.269,Z 764.97,A -85,B 0,C 180,E1 25541.459,E2 25541.459} C_VEL
LIN {X 0,Y 538.403,Z 748.328,A -85,B 0,C 180,E1 25541.014,E2 25541.014} C_VEL
LIN {X 0,Y 539.767,Z 611.553,A -85,B 0,C 180,E1 25538.914,E2 25538.914} C_VEL
LIN {X 0,Y 540.338,Z 607.186,A -85,B 0,C 180,E1 25538.507,E2 25538.507} C_VEL
LIN {X 0,Y 542.495,Z 571.229,A -85,B 0,C 180,E1 25534.855,E2 25534.855} C_VEL
LIN {X 0,Y 545.474,Z 537.328,A -85,B 0,C 180,E1 25531.239,E2 25531.239} C_VEL
LIN {X 0,Y 549.12,Z 508.857,A -85,B 0,C 180,E1 25528.004,E2 25528.004} C_VEL
LIN {X 0,Y 551.331,Z 495.3,A -85,B 0,C 180,E1 25526.348,E2 25526.348} C_VEL
LIN {X 0,Y 553.344,Z 483.217,A -85,B 0,C 180,E1 25524.675,E2 25524.675} C_VEL
LIN {X 0,Y 551.661,Z 477.737,A -85,B 0,C 180,E1 25523.063,E2 25523.063} C_VEL
LIN {X 0,Y 550.687,Z 474.43,A -85,B 0,C 180,E1 25521.481,E2 25521.481} C_VEL
LIN {X 0,Y 550.446,Z 473.845,A -85,B 0,C 180,E1 25520.118,E2 25520.118} C_VEL
LIN {X 0,Y 551.236,Z 474.821,A -85,B 0,C 180,E1 25518.958,E2 25518.958} C_VEL
LIN {X 0,Y 551.77,Z 476.592,A -85,B 0,C 180,E1 25518.296,E2 25518.296} C_VEL
LIN {X 0,Y 552.259,Z 478.211,A -85,B 0,C 180,E1 25517.851,E2 25517.851} C_VEL
LIN {X 0,Y 548.636,Z 492.579,A -85,B 0,C 180,E1 25516.497,E2 25516.497} C_VEL
LIN {X 0,Y 545.531,Z 512.906,A -85,B 0,C 180,E1 25514.822,E2 25514.822} C_VEL
LIN {X 0,Y 543.292,Z 540.497,A -85,B 0,C 180,E1 25512.774,E2 25512.774} C_VEL
LIN {X 0,Y 543.634,Z 559.486,A -85,B 0,C 180,E1 25511.375,E2 25511.375} C_VEL
LIN {X 0,Y 545.631,Z 573.359,A -85,B 0,C 180,E1 25510.306,E2 25510.306} C_VEL
LIN {X 0,Y 549.439,Z 585.707,A -85,B 0,C 180,E1 25509.294,E2 25509.294} C_VEL
LIN {X 0,Y 554.262,Z 595.039,A -85,B 0,C 180,E1 25508.472,E2 25508.472} C_VEL
LIN {X 0,Y 560.118,Z 602.701,A -85,B 0,C 180,E1 25507.741,E2 25507.741} C_VEL
LIN {X 0,Y 567.369,Z 609.39,A -85,B 0,C 180,E1 25507.031,E2 25507.031} C_VEL
LIN {X 0,Y 575.163,Z 614.445,A -85,B 0,C 180,E1 25506.402,E2 25506.402} C_VEL
LIN {X 0,Y 579.452,Z 616.178,A -85,B 0,C 180,E1 25505.975,E2 25505.975} C_VEL
LIN {X 0,Y 583.143,Z 616.781,A -85,B 0,C 180,E1 25505.469,E2 25505.469} C_VEL
LIN {X 0,Y 585.667,Z 616.32,A -85,B 0,C 180,E1 25504.969,E2 25504.969} C_VEL
LIN {X 0,Y 587.414,Z 614.687,A -85,B 0,C 180,E1 25504.357,E2 25504.357} C_VEL
LIN {X 0,Y 587.7,Z 612.052,A -85,B 0,C 180,E1 25503.773,E2 25503.773} C_VEL
LIN {X 0,Y 586.43,Z 608.341,A -85,B 0,C 180,E1 25503.212,E2 25503.212} C_VEL
LIN {X 0,Y 582.933,Z 602.582,A -85,B 0,C 180,E1 25502.617,E2 25502.617} C_VEL
LIN {X 0,Y 578.263,Z 593.081,A -85,B 0,C 180,E1 25501.887,E2 25501.887} C_VEL
LIN {X 0,Y 575.997,Z 587.303,A -85,B 0,C 180,E1 25501.522,E2 25501.522} C_VEL
LIN {X 0,Y 571.473,Z 644.088,A -85,B 0,C 180,E1 25500.775,E2 25500.775} C_VEL
LIN {X 0,Y 568.567,Z 670.138,A -85,B 0,C 180,E1 25500.36,E2 25500.36} C_VEL
LIN {X 0,Y 565.244,Z 687.292,A -85,B 0,C 180,E1 25500.018,E2 25500.018} C_VEL
LIN {X 0,Y 563.426,Z 694.755,A -85,B 0,C 180,E1 25499.782,E2 25499.782} C_VEL
LIN {X 0,Y 558.935,Z 712.332,A -85,B 0,C 180,E1 25499.645,E2 25499.645} C_VEL
LIN {X 0,Y 553.779,Z 728.086,A -85,B 0,C 180,E1 25499.384,E2 25499.384} C_VEL
LIN {X 0,Y 549.738,Z 740.438,A -85,B 0,C 180,E1 25498.994,E2 25498.994} C_VEL
LIN {X 0,Y 547.839,Z 747.143,A -85,B 0,C 180,E1 25498.686,E2 25498.686} C_VEL
LIN {X 0,Y 544.628,Z 756.994,A -85,B 0,C 180,E1 25498.332,E2 25498.332} C_VEL
LIN {X 0,Y 543.336,Z 762.694,A -85,B 0,C 180,E1 25498.065,E2 25498.065} C_VEL
LIN {X 0,Y 542.921,Z 807.578,A -85,B 0,C 180,E1 25497.392,E2 25497.392} C_VEL
LIN {X 0,Y 542.45,Z 828.761,A -85,B 0,C 180,E1 25496.873,E2 25496.873} C_VEL
LIN {X 0,Y 541.854,Z 849.051,A -85,B 0,C 180,E1 25496.169,E2 25496.169} C_VEL
LIN {X 0,Y 541.155,Z 868.877,A -85,B 0,C 180,E1 25495.266,E2 25495.266} C_VEL
LIN {X 0,Y 540.397,Z 887.802,A -85,B 0,C 180,E1 25494.194,E2 25494.194} C_VEL
LIN {X 0,Y 539.605,Z 905.957,A -85,B 0,C 180,E1 25492.94,E2 25492.94} C_VEL
LIN {X 0,Y 538.802,Z 924.041,A -85,B 0,C 180,E1 25491.444,E2 25491.444} C_VEL
LIN {X 0,Y 538.074,Z 940.374,A -85,B 0,C 180,E1 25489.824,E2 25489.824} C_VEL
LIN {X 0,Y 537.496,Z 954.316,A -85,B 0,C 180,E1 25488.212,E2 25488.212} C_VEL
LIN {X 0,Y 536.962,Z 968.069,A -85,B 0,C 180,E1 25486.331,E2 25486.331} C_VEL
LIN {X 0,Y 536.575,Z 979.657,A -85,B 0,C 180,E1 25484.46,E2 25484.46} C_VEL
LIN {X 0,Y 536.28,Z 990.36,A -85,B 0,C 180,E1 25482.381,E2 25482.381} C_VEL
LIN {X 0,Y 536.089,Z 999.093,A -85,B 0,C 180,E1 25480.315,E2 25480.315} C_VEL
LIN {X 0,Y 535.985,Z 1006.279,A -85,B 0,C 180,E1 25478.151,E2 25478.151} C_VEL
LIN {X 0,Y 535.938,Z 1011.735,A -85,B 0,C 180,E1 25475.997,E2 25475.997} C_VEL
LIN {X 0,Y 535.913,Z 1015.527,A -85,B 0,C 180,E1 25473.745,E2 25473.745} C_VEL
LIN {X 0,Y 535.902,Z 1017.526,A -85,B 0,C 180,E1 25471.604,E2 25471.604} C_VEL
LIN {X 0,Y 535.902,Z 1017.871,A -85,B 0,C 180,E1 25469.359,E2 25469.359} C_VEL
LIN {X 0,Y 535.912,Z 1016.644,A -85,B 0,C 180,E1 25467.22,E2 25467.22} C_VEL
LIN {X 0,Y 535.916,Z 1013.556,A -85,B 0,C 180,E1 25464.97,E2 25464.97} C_VEL
LIN {X 0,Y 535.943,Z 1009.217,A -85,B 0,C 180,E1 25462.928,E2 25462.928} C_VEL
LIN {X 0,Y 536.02,Z 1002.939,A -85,B 0,C 180,E1 25460.769,E2 25460.769} C_VEL
LIN {X 0,Y 536.177,Z 994.75,A -85,B 0,C 180,E1 25458.6,E2 25458.6} C_VEL
LIN {X 0,Y 536.417,Z 984.973,A -85,B 0,C 180,E1 25456.527,E2 25456.527} C_VEL
LIN {X 0,Y 536.745,Z 974.481,A -85,B 0,C 180,E1 25454.662,E2 25454.662} C_VEL
LIN {X 0,Y 537.216,Z 961.294,A -85,B 0,C 180,E1 25452.705,E2 25452.705} C_VEL
LIN {X 0,Y 537.758,Z 947.888,A -85,B 0,C 180,E1 25451.012,E2 25451.012} C_VEL
LIN {X 0,Y 538.423,Z 932.267,A -85,B 0,C 180,E1 25449.34,E2 25449.34} C_VEL
LIN {X 0,Y 539.143,Z 916.332,A -85,B 0,C 180,E1 25447.885,E2 25447.885} C_VEL
LIN {X 0,Y 539.966,Z 898.01,A -85,B 0,C 180,E1 25446.482,E2 25446.482} C_VEL
LIN {X 0,Y 540.742,Z 879.349,A -85,B 0,C 180,E1 25445.299,E2 25445.299} C_VEL
LIN {X 0,Y 541.489,Z 859.583,A -85,B 0,C 180,E1 25444.284,E2 25444.284} C_VEL
LIN {X 0,Y 542.159,Z 839.26,A -85,B 0,C 180,E1 25443.463,E2 25443.463} C_VEL
LIN {X 0,Y 542.705,Z 818.455,A -85,B 0,C 180,E1 25442.849,E2 25442.849} C_VEL
LIN {X 0,Y 543.067,Z 796.939,A -85,B 0,C 180,E1 25442.424,E2 25442.424} C_VEL
LIN {X 0,Y 543.435,Z 761.553,A -85,B 0,C 180,E1 25441.901,E2 25441.901} C_VEL
LIN {X 0,Y 545.865,Z 752.948,A -85,B 0,C 180,E1 25441.501,E2 25441.501} C_VEL
LIN {X 0,Y 548.388,Z 745.225,A -85,B 0,C 180,E1 25441.228,E2 25441.228} C_VEL
LIN {X 0,Y 551.452,Z 735.018,A -85,B 0,C 180,E1 25440.809,E2 25440.809} C_VEL
LIN {X 0,Y 556.158,Z 721.043,A -85,B 0,C 180,E1 25440.474,E2 25440.474} C_VEL
LIN {X 0,Y 561.327,Z 703.817,A -85,B 0,C 180,E1 25440.278,E2 25440.278} C_VEL
LIN {X 0,Y 563.795,Z 693.133,A -85,B 0,C 180,E1 25440.184,E2 25440.184} C_VEL
LIN {X 0,Y 566.06,Z 683.638,A -85,B 0,C 180,E1 25439.892,E2 25439.892} C_VEL
LIN {X 0,Y 569.493,Z 663.68,A -85,B 0,C 180,E1 25439.536,E2 25439.536} C_VEL
LIN {X 0,Y 573.474,Z 620.417,A -85,B 0,C 180,E1 25438.891,E2 25438.891} C_VEL
LIN {X 0,Y 576.09,Z 587.313,A -85,B 0,C 180,E1 25438.463,E2 25438.463} C_VEL
LIN {X 0,Y 580.18,Z 597.37,A -85,B 0,C 180,E1 25437.81,E2 25437.81} C_VEL
LIN {X 0,Y 585.022,Z 605.931,A -85,B 0,C 180,E1 25437.064,E2 25437.064} C_VEL
LIN {X 0,Y 587.137,Z 609.91,A -85,B 0,C 180,E1 25436.572,E2 25436.572} C_VEL
LIN {X 0,Y 587.757,Z 613.232,A -85,B 0,C 180,E1 25435.997,E2 25435.997} C_VEL
LIN {X 0,Y 586.842,Z 615.518,A -85,B 0,C 180,E1 25435.379,E2 25435.379} C_VEL
LIN {X 0,Y 584.658,Z 616.653,A -85,B 0,C 180,E1 25434.808,E2 25434.808} C_VEL
LIN {X 0,Y 581.378,Z 616.62,A -85,B 0,C 180,E1 25434.267,E2 25434.267} C_VEL
LIN {X 0,Y 577.376,Z 615.461,A -85,B 0,C 180,E1 25433.802,E2 25433.802} C_VEL
LIN {X 0,Y 569.503,Z 611.173,A -85,B 0,C 180,E1 25433.018,E2 25433.018} C_VEL
LIN {X 0,Y 562.303,Z 605.114,A -85,B 0,C 180,E1 25432.138,E2 25432.138} C_VEL
LIN {X 0,Y 556.533,Z 597.703,A -85,B 0,C 180,E1 25431.234,E2 25431.234} C_VEL
LIN {X 0,Y 552.186,Z 588.973,A -85,B 0,C 180,E1 25430.314,E2 25430.314} C_VEL
LIN {X 0,Y 548.929,Z 577.614,A -85,B 0,C 180,E1 25429.264,E2 25429.264} C_VEL
LIN {X 0,Y 547.169,Z 563.878,A -85,B 0,C 180,E1 25428.136,E2 25428.136} C_VEL
LIN {X 0,Y 546.986,Z 544.257,A -85,B 0,C 180,E1 25426.679,E2 25426.679} C_VEL
LIN {X 0,Y 548.748,Z 505.489,A -85,B 0,C 180,E1 25423.819,E2 25423.819} C_VEL
LIN {X 0,Y 549.923,Z 476.82,A -85,B 0,C 180,E1 25421.623,E2 25421.623} C_VEL
LIN {X 0,Y 541.853,Z 460.352,A -85,B 0,C 180,E1 25419.403,E2 25419.403} C_VEL
LIN {X 0,Y 537.804,Z 452.197,A -85,B 0,C 180,E1 25418.25,E2 25418.25} C_VEL
LIN {X 0,Y 536.443,Z 448.666,A -85,B 0,C 180,E1 25417.746,E2 25417.746} C_VEL
LIN {X 0,Y 536.468,Z 448.657,A -85,B 0,C 180,E1 25414.254,E2 25414.254} C_VEL
LIN {X 0,Y 536.437,Z 448.665,A -85,B 0,C 180,E1 25410.835,E2 25410.835} C_VEL
LIN {X 0,Y 536.421,Z 448.666,A -85,B 0,C 180,E1 25407.412,E2 25407.412} C_VEL
LIN {X 0,Y 536.456,Z 448.663,A -85,B 0,C 180,E1 25404.207,E2 25404.207} C_VEL
LIN {X 0,Y 536.415,Z 448.667,A -85,B 0,C 180,E1 25400.741,E2 25400.741} C_VEL
LIN {X 0,Y 536.45,Z 448.662,A -85,B 0,C 180,E1 25397.35,E2 25397.35} C_VEL
LIN {X 0,Y 536.436,Z 448.664,A -85,B 0,C 180,E1 25394.022,E2 25394.022} C_VEL
LIN {X 0,Y 536.411,Z 448.667,A -85,B 0,C 180,E1 25390.525,E2 25390.525} C_VEL
LIN {X 0,Y 536.465,Z 448.659,A -85,B 0,C 180,E1 25387.173,E2 25387.173} C_VEL
LIN {X 0,Y 536.411,Z 448.666,A -85,B 0,C 180,E1 25383.847,E2 25383.847} C_VEL
LIN {X 0,Y 536.437,Z 448.661,A -85,B 0,C 180,E1 25380.427,E2 25380.427} C_VEL
LIN {X 0,Y 536.45,Z 448.661,A -85,B 0,C 180,E1 25377.115,E2 25377.115} C_VEL
LIN {X 0,Y 536.416,Z 448.665,A -85,B 0,C 180,E1 25373.686,E2 25373.686} C_VEL
LIN {X 0,Y 536.457,Z 448.66,A -85,B 0,C 180,E1 25370.235,E2 25370.235} C_VEL
LIN {X 0,Y 536.424,Z 448.66,A -85,B 0,C 180,E1 25366.965,E2 25366.965} C_VEL
LIN {X 0,Y 536.438,Z 448.663,A -85,B 0,C 180,E1 25363.653,E2 25363.653} C_VEL
LIN {X 0,Y 536.466,Z 448.659,A -85,B 0,C 180,E1 25360.255,E2 25360.255} C_VEL
LIN {X 0,Y 536.433,Z 448.659,A -85,B 0,C 180,E1 25356.841,E2 25356.841} C_VEL
LIN {X 0,Y 536.46,Z 448.661,A -85,B 0,C 180,E1 25353.428,E2 25353.428} C_VEL
LIN {X 0,Y 536.461,Z 448.664,A -85,B 0,C 180,E1 25350.033,E2 25350.033} C_VEL
LIN {X 0,Y 536.461,Z 448.665,A -85,B 0,C 180,E1 25346.613,E2 25346.613} C_VEL
LIN {X 0,Y 536.454,Z 448.66,A -85,B 0,C 180,E1 25345.379,E2 25345.379} C_VEL
LIN {X 0,Y 535.476,Z 448.787,A -85,B 0,C 180,E1 25344.556,E2 25344.556} C_VEL
LIN {X 0,Y 528.986,Z 449.59,A -85,B 0,C 180,E1 25342.186,E2 25342.186} C_VEL
LIN {X 0,Y 528.521,Z 449.65,A -85,B 0,C 180,E1 25341.643,E2 25341.643} C_VEL
LIN {X 0,Y 528.527,Z 449.652,A -85,B 0,C 180,E1 25338.189,E2 25338.189} C_VEL
LIN {X 0,Y 528.5,Z 449.654,A -85,B 0,C 180,E1 25334.73,E2 25334.73} C_VEL
LIN {X 0,Y 528.524,Z 449.653,A -85,B 0,C 180,E1 25331.317,E2 25331.317} C_VEL
LIN {X 0,Y 528.507,Z 449.655,A -85,B 0,C 180,E1 25327.916,E2 25327.916} C_VEL
LIN {X 0,Y 528.492,Z 449.707,A -85,B 0,C 180,E1 25326.146,E2 25326.146} C_VEL
LIN {X 0,Y 536.273,Z 471.172,A -85,B 0,C 180,E1 25323.742,E2 25323.742} C_VEL
LIN {X 0,Y 535.546,Z 495.83,A -85,B 0,C 180,E1 25321.766,E2 25321.766} C_VEL
LIN {X 0,Y 538.085,Z 510.174,A -85,B 0,C 180,E1 25321.376,E2 25321.376} C_VEL
LIN {X 0,Y 535.846,Z 755.49,A -85,B 0,C 180,E1 25317.779,E2 25317.779} C_VEL
LIN {X 0,Y 535.328,Z 776.497,A -85,B 0,C 180,E1 25317.281,E2 25317.281} C_VEL
LIN {X 0,Y 534.686,Z 797.17,A -85,B 0,C 180,E1 25316.576,E2 25316.576} C_VEL
LIN {X 0,Y 533.926,Z 816.922,A -85,B 0,C 180,E1 25315.69,E2 25315.69} C_VEL
LIN {X 0,Y 533.099,Z 835.304,A -85,B 0,C 180,E1 25314.664,E2 25314.664} C_VEL
LIN {X 0,Y 532.239,Z 853.714,A -85,B 0,C 180,E1 25313.41,E2 25313.41} C_VEL
LIN {X 0,Y 531.362,Z 871.047,A -85,B 0,C 180,E1 25311.99,E2 25311.99} C_VEL
LIN {X 0,Y 530.561,Z 886.768,A -85,B 0,C 180,E1 25310.467,E2 25310.467} C_VEL
LIN {X 0,Y 529.857,Z 901.239,A -85,B 0,C 180,E1 25308.825,E2 25308.825} C_VEL
LIN {X 0,Y 529.222,Z 915.521,A -85,B 0,C 180,E1 25306.914,E2 25306.914} C_VEL
LIN {X 0,Y 528.727,Z 928.143,A -85,B 0,C 180,E1 25304.903,E2 25304.903} C_VEL
LIN {X 0,Y 528.374,Z 939.141,A -85,B 0,C 180,E1 25302.791,E2 25302.791} C_VEL
LIN {X 0,Y 528.142,Z 948.098,A -85,B 0,C 180,E1 25300.691,E2 25300.691} C_VEL
LIN {X 0,Y 528.014,Z 955.572,A -85,B 0,C 180,E1 25298.493,E2 25298.493} C_VEL
LIN {X 0,Y 527.945,Z 961.151,A -85,B 0,C 180,E1 25296.306,E2 25296.306} C_VEL
LIN {X 0,Y 527.92,Z 965.018,A -85,B 0,C 180,E1 25294.127,E2 25294.127} C_VEL
LIN {X 0,Y 527.912,Z 967.346,A -85,B 0,C 180,E1 25291.845,E2 25291.845} C_VEL
LIN {X 0,Y 527.904,Z 967.949,A -85,B 0,C 180,E1 25289.674,E2 25289.674} C_VEL
LIN {X 0,Y 527.905,Z 966.991,A -85,B 0,C 180,E1 25287.503,E2 25287.503} C_VEL
LIN {X 0,Y 527.921,Z 964.357,A -85,B 0,C 180,E1 25285.328,E2 25285.328} C_VEL
LIN {X 0,Y 527.953,Z 960.094,A -85,B 0,C 180,E1 25283.147,E2 25283.147} C_VEL
LIN {X 0,Y 528.022,Z 954.115,A -85,B 0,C 180,E1 25280.957,E2 25280.957} C_VEL
LIN {X 0,Y 528.165,Z 946.728,A -85,B 0,C 180,E1 25278.866,E2 25278.866} C_VEL
LIN {X 0,Y 528.425,Z 937.48,A -85,B 0,C 180,E1 25276.764,E2 25276.764} C_VEL
LIN {X 0,Y 528.784,Z 926.734,A -85,B 0,C 180,E1 25274.761,E2 25274.761} C_VEL
LIN {X 0,Y 529.26,Z 914.594,A -85,B 0,C 180,E1 25272.859,E2 25272.859} C_VEL
LIN {X 0,Y 529.903,Z 900.272,A -85,B 0,C 180,E1 25270.966,E2 25270.966} C_VEL
LIN {X 0,Y 530.644,Z 884.931,A -85,B 0,C 180,E1 25269.253,E2 25269.253} C_VEL
LIN {X 0,Y 531.492,Z 868.109,A -85,B 0,C 180,E1 25267.665,E2 25267.665} C_VEL
LIN {X 0,Y 532.4,Z 850.144,A -85,B 0,C 180,E1 25266.244,E2 25266.244} C_VEL
LIN {X 0,Y 533.253,Z 831.968,A -85,B 0,C 180,E1 25265.046,E2 25265.046} C_VEL
LIN {X 0,Y 534.085,Z 812.926,A -85,B 0,C 180,E1 25264.019,E2 25264.019} C_VEL
LIN {X 0,Y 534.861,Z 792.814,A -85,B 0,C 180,E1 25263.162,E2 25263.162} C_VEL
LIN {X 0,Y 535.479,Z 772.095,A -85,B 0,C 180,E1 25262.504,E2 25262.504} C_VEL
LIN {X 0,Y 535.908,Z 751.439,A -85,B 0,C 180,E1 25262.057,E2 25262.057} C_VEL
LIN {X 0,Y 537.973,Z 514.455,A -85,B 0,C 180,E1 25258.592,E2 25258.592} C_VEL
LIN {X 0,Y 533.458,Z 497.842,A -85,B 0,C 180,E1 25258.022,E2 25258.022} C_VEL
LIN {X 0,Y 534.422,Z 473.432,A -85,B 0,C 180,E1 25255.031,E2 25255.031} C_VEL
LIN {X 0,Y 534.309,Z 468.536,A -85,B 0,C 180,E1 25254.41,E2 25254.41} C_VEL
LIN {X 0,Y 529.191,Z 452.088,A -85,B 0,C 180,E1 25251.901,E2 25251.901} C_VEL
LIN {X 0,Y 528.503,Z 449.659,A -85,B 0,C 180,E1 25251.506,E2 25251.506} C_VEL
LIN {X 0,Y 528.493,Z 449.653,A -85,B 0,C 180,E1 25248.098,E2 25248.098} C_VEL
LIN {X 0,Y 528.524,Z 449.647,A -85,B 0,C 180,E1 25244.729,E2 25244.729} C_VEL
LIN {X 0,Y 528.521,Z 449.65,A -85,B 0,C 180,E1 25241.318,E2 25241.318} C_VEL
LIN {X 0,Y 528.512,Z 449.65,A -85,B 0,C 180,E1 25237.917,E2 25237.917} C_VEL
LIN {X 0,Y 528.509,Z 449.654,A -85,B 0,C 180,E1 25234.58,E2 25234.58} C_VEL
LIN {X 0,Y 528.522,Z 449.659,A -85,B 0,C 180,E1 25231.095,E2 25231.095} C_VEL
LIN {X 0,Y 528.521,Z 449.722,A -85,B 0,C 180,E1 25230.969,E2 25230.969} C_VEL
LIN {X 0,Y 535.364,Z 470.182,A -85,B 0,C 180,E1 25228.354,E2 25228.354} C_VEL
LIN {X 0,Y 534.334,Z 501.798,A -85,B 0,C 180,E1 25225.255,E2 25225.255} C_VEL
LIN {X 0,Y 533.204,Z 536.503,A -85,B 0,C 180,E1 25221.911,E2 25221.911} C_VEL
LIN {X 0,Y 532.039,Z 572.209,A -85,B 0,C 180,E1 25218.518,E2 25218.518} C_VEL
LIN {X 0,Y 531.202,Z 607.164,A -85,B 0,C 180,E1 25215.266,E2 25215.266} C_VEL
LIN {X 0,Y 531.786,Z 613.232,A -85,B 0,C 180,E1 25215.145,E2 25215.145} C_VEL
LIN {X 0,Y 530.703,Z 748.838,A -85,B 0,C 180,E1 25213.12,E2 25213.12} C_VEL
LIN {X 0,Y 530.515,Z 765.503,A -85,B 0,C 180,E1 25212.656,E2 25212.656} C_VEL
LIN {X 0,Y 530.25,Z 780.694,A -85,B 0,C 180,E1 25212.027,E2 25212.027} C_VEL
LIN {X 0,Y 529.895,Z 796.258,A -85,B 0,C 180,E1 25211.152,E2 25211.152} C_VEL
LIN {X 0,Y 529.526,Z 809.651,A -85,B 0,C 180,E1 25210.169,E2 25210.169} C_VEL
LIN {X 0,Y 529.143,Z 822.713,A -85,B 0,C 180,E1 25208.969,E2 25208.969} C_VEL
LIN {X 0,Y 528.816,Z 833.568,A -85,B 0,C 180,E1 25207.715,E2 25207.715} C_VEL
LIN {X 0,Y 528.557,Z 842.772,A -85,B 0,C 180,E1 25206.408,E2 25206.408} C_VEL
LIN {X 0,Y 528.345,Z 851.397,A -85,B 0,C 180,E1 25204.885,E2 25204.885} C_VEL
LIN {X 0,Y 528.191,Z 858.416,A -85,B 0,C 180,E1 25203.256,E2 25203.256} C_VEL
LIN {X 0,Y 528.102,Z 863.663,A -85,B 0,C 180,E1 25201.628,E2 25201.628} C_VEL
LIN {X 0,Y 528.058,Z 867.596,A -85,B 0,C 180,E1 25199.783,E2 25199.783} C_VEL
LIN {X 0,Y 528.041,Z 869.486,A -85,B 0,C 180,E1 25198.047,E2 25198.047} C_VEL
LIN {X 0,Y 528.046,Z 869.802,A -85,B 0,C 180,E1 25196.276,E2 25196.276} C_VEL
LIN {X 0,Y 528.068,Z 868.352,A -85,B 0,C 180,E1 25194.568,E2 25194.568} C_VEL
LIN {X 0,Y 528.114,Z 865.515,A -85,B 0,C 180,E1 25192.931,E2 25192.931} C_VEL
LIN {X 0,Y 528.221,Z 860.622,A -85,B 0,C 180,E1 25191.15,E2 25191.15} C_VEL
LIN {X 0,Y 528.379,Z 854.284,A -85,B 0,C 180,E1 25189.534,E2 25189.534} C_VEL
LIN {X 0,Y 528.591,Z 846.503,A -85,B 0,C 180,E1 25187.991,E2 25187.991} C_VEL
LIN {X 0,Y 528.905,Z 836.363,A -85,B 0,C 180,E1 25186.443,E2 25186.443} C_VEL
LIN {X 0,Y 529.273,Z 825.151,A -85,B 0,C 180,E1 25185.084,E2 25185.084} C_VEL
LIN {X 0,Y 529.689,Z 812.047,A -85,B 0,C 180,E1 25183.834,E2 25183.834} C_VEL
LIN {X 0,Y 530.05,Z 799.108,A -85,B 0,C 180,E1 25182.854,E2 25182.854} C_VEL
LIN {X 0,Y 530.357,Z 784.311,A -85,B 0,C 180,E1 25181.99,E2 25181.99} C_VEL
LIN {X 0,Y 530.606,Z 769.636,A -85,B 0,C 180,E1 25181.348,E2 25181.348} C_VEL
LIN {X 0,Y 530.724,Z 753.785,A -85,B 0,C 180,E1 25180.876,E2 25180.876} C_VEL
LIN {X 0,Y 530.871,Z 729.467,A -85,B 0,C 180,E1 25180.463,E2 25180.463} C_VEL
LIN {X 0,Y 532.334,Z 618.589,A -85,B 0,C 180,E1 25178.683,E2 25178.683} C_VEL
LIN {X 0,Y 532.515,Z 613.877,A -85,B 0,C 180,E1 25178.581,E2 25178.581} C_VEL
LIN {X 0,Y 533.218,Z 610.87,A -85,B 0,C 180,E1 25178.321,E2 25178.321} C_VEL
LIN {X 0,Y 535.667,Z 574.59,A -85,B 0,C 180,E1 25174.576,E2 25174.576} C_VEL
LIN {X 0,Y 538.997,Z 540.751,A -85,B 0,C 180,E1 25170.895,E2 25170.895} C_VEL
LIN {X 0,Y 542.933,Z 513.283,A -85,B 0,C 180,E1 25167.704,E2 25167.704} C_VEL
LIN {X 0,Y 545.566,Z 499.178,A -85,B 0,C 180,E1 25165.934,E2 25165.934} C_VEL
LIN {X 0,Y 547.683,Z 488.358,A -85,B 0,C 180,E1 25164.383,E2 25164.383} C_VEL
LIN {X 0,Y 546.297,Z 483.378,A -85,B 0,C 180,E1 25162.766,E2 25162.766} C_VEL
LIN {X 0,Y 545.82,Z 480.777,A -85,B 0,C 180,E1 25161.463,E2 25161.463} C_VEL
LIN {X 0,Y 545.694,Z 480.28,A -85,B 0,C 180,E1 25160.112,E2 25160.112} C_VEL
LIN {X 0,Y 546.587,Z 481.38,A -85,B 0,C 180,E1 25158.888,E2 25158.888} C_VEL
LIN {X 0,Y 546.93,Z 483.466,A -85,B 0,C 180,E1 25158.235,E2 25158.235} C_VEL
LIN {X 0,Y 542.885,Z 497.003,A -85,B 0,C 180,E1 25156.899,E2 25156.899} C_VEL
LIN {X 0,Y 539.418,Z 515.312,A -85,B 0,C 180,E1 25155.305,E2 25155.305} C_VEL
LIN {X 0,Y 536.72,Z 540.225,A -85,B 0,C 180,E1 25153.36,E2 25153.36} C_VEL
LIN {X 0,Y 536.519,Z 559.625,A -85,B 0,C 180,E1 25151.875,E2 25151.875} C_VEL
LIN {X 0,Y 538.188,Z 574.474,A -85,B 0,C 180,E1 25150.701,E2 25150.701} C_VEL
LIN {X 0,Y 541.766,Z 587.56,A -85,B 0,C 180,E1 25149.6,E2 25149.6} C_VEL
LIN {X 0,Y 546.45,Z 597.551,A -85,B 0,C 180,E1 25148.705,E2 25148.705} C_VEL
LIN {X 0,Y 552.404,Z 606.021,A -85,B 0,C 180,E1 25147.893,E2 25147.893} C_VEL
LIN {X 0,Y 560.206,Z 613.787,A -85,B 0,C 180,E1 25147.079,E2 25147.079} C_VEL
LIN {X 0,Y 569.533,Z 620.21,A -85,B 0,C 180,E1 25146.312,E2 25146.312} C_VEL
LIN {X 0,Y 574.998,Z 622.791,A -85,B 0,C 180,E1 25145.873,E2 25145.873} C_VEL
LIN {X 0,Y 579.071,Z 623.809,A -85,B 0,C 180,E1 25145.415,E2 25145.415} C_VEL
LIN {X 0,Y 582.5,Z 623.704,A -85,B 0,C 180,E1 25144.862,E2 25144.862} C_VEL
LIN {X 0,Y 584.648,Z 622.545,A -85,B 0,C 180,E1 25144.308,E2 25144.308} C_VEL
LIN {X 0,Y 585.599,Z 620.308,A -85,B 0,C 180,E1 25143.705,E2 25143.705} C_VEL
LIN {X 0,Y 585.023,Z 616.984,A -85,B 0,C 180,E1 25143.117,E2 25143.117} C_VEL
LIN {X 0,Y 582.929,Z 613.08,A -85,B 0,C 180,E1 25142.617,E2 25142.617} C_VEL
LIN {X 0,Y 578.809,Z 606.528,A -85,B 0,C 180,E1 25141.973,E2 25141.973} C_VEL
LIN {X 0,Y 575.262,Z 645.647,A -85,B 0,C 180,E1 25141.462,E2 25141.462} C_VEL
LIN {X 0,Y 571.357,Z 666.878,A -85,B 0,C 180,E1 25141.198,E2 25141.198} C_VEL
LIN {X 0,Y 566.235,Z 686.155,A -85,B 0,C 180,E1 25140.88,E2 25140.88} C_VEL
LIN {X 0,Y 563.325,Z 695.977,A -85,B 0,C 180,E1 25140.589,E2 25140.589} C_VEL
LIN {X 0,Y 556.689,Z 713.575,A -85,B 0,C 180,E1 25140.431,E2 25140.431} C_VEL
LIN {X 0,Y 550.267,Z 728.651,A -85,B 0,C 180,E1 25140.128,E2 25140.128} C_VEL
LIN {X 0,Y 545.599,Z 740.679,A -85,B 0,C 180,E1 25139.718,E2 25139.718} C_VEL
LIN {X 0,Y 542.835,Z 749.247,A -85,B 0,C 180,E1 25139.338,E2 25139.338} C_VEL
LIN {X 0,Y 539.347,Z 758.994,A -85,B 0,C 180,E1 25138.938,E2 25138.938} C_VEL
LIN {X 0,Y 536.208,Z 771.028,A -85,B 0,C 180,E1 25138.348,E2 25138.348} C_VEL
LIN {X 0,Y 535.798,Z 808.27,A -85,B 0,C 180,E1 25137.772,E2 25137.772} C_VEL
LIN {X 0,Y 535.273,Z 829.452,A -85,B 0,C 180,E1 25137.242,E2 25137.242} C_VEL
LIN {X 0,Y 534.598,Z 849.723,A -85,B 0,C 180,E1 25136.522,E2 25136.522} C_VEL
LIN {X 0,Y 533.8,Z 869.987,A -85,B 0,C 180,E1 25135.579,E2 25135.579} C_VEL
LIN {X 0,Y 532.953,Z 888.7,A -85,B 0,C 180,E1 25134.496,E2 25134.496} C_VEL
LIN {X 0,Y 532.046,Z 907.121,A -85,B 0,C 180,E1 25133.192,E2 25133.192} C_VEL
LIN {X 0,Y 531.185,Z 924.475,A -85,B 0,C 180,E1 25131.726,E2 25131.726} C_VEL
LIN {X 0,Y 530.397,Z 940.115,A -85,B 0,C 180,E1 25130.152,E2 25130.152} C_VEL
LIN {X 0,Y 529.76,Z 953.394,A -85,B 0,C 180,E1 25128.601,E2 25128.601} C_VEL
LIN {X 0,Y 529.142,Z 967.529,A -85,B 0,C 180,E1 25126.661,E2 25126.661} C_VEL
LIN {X 0,Y 528.693,Z 979.018,A -85,B 0,C 180,E1 25124.793,E2 25124.793} C_VEL
LIN {X 0,Y 528.354,Z 989.852,A -85,B 0,C 180,E1 25122.681,E2 25122.681} C_VEL
LIN {X 0,Y 528.132,Z 998.69,A -85,B 0,C 180,E1 25120.582,E2 25120.582} C_VEL
LIN {X 0,Y 528.004,Z 1005.965,A -85,B 0,C 180,E1 25118.385,E2 25118.385} C_VEL
LIN {X 0,Y 527.944,Z 1011.233,A -85,B 0,C 180,E1 25116.307,E2 25116.307} C_VEL
LIN {X 0,Y 527.92,Z 1015.248,A -85,B 0,C 180,E1 25114.019,E2 25114.019} C_VEL
LIN {X 0,Y 527.91,Z 1017.395,A -85,B 0,C 180,E1 25111.846,E2 25111.846} C_VEL
LIN {X 0,Y 527.9,Z 1017.918,A -85,B 0,C 180,E1 25109.566,E2 25109.566} C_VEL
LIN {X 0,Y 527.908,Z 1016.912,A -85,B 0,C 180,E1 25107.504,E2 25107.504} C_VEL
LIN {X 0,Y 527.922,Z 1014.137,A -85,B 0,C 180,E1 25105.22,E2 25105.22} C_VEL
LIN {X 0,Y 527.951,Z 1009.975,A -85,B 0,C 180,E1 25103.148,E2 25103.148} C_VEL
LIN {X 0,Y 528.022,Z 1004.006,A -85,B 0,C 180,E1 25100.958,E2 25100.958} C_VEL
LIN {X 0,Y 528.167,Z 996.523,A -85,B 0,C 180,E1 25098.867,E2 25098.867} C_VEL
LIN {X 0,Y 528.434,Z 987.268,A -85,B 0,C 180,E1 25096.766,E2 25096.766} C_VEL
LIN {X 0,Y 528.788,Z 976.433,A -85,B 0,C 180,E1 25094.763,E2 25094.763} C_VEL
LIN {X 0,Y 529.313,Z 963.536,A -85,B 0,C 180,E1 25092.749,E2 25092.749} C_VEL
LIN {X 0,Y 529.925,Z 949.733,A -85,B 0,C 180,E1 25090.949,E2 25090.949} C_VEL
LIN {X 0,Y 530.695,Z 933.976,A -85,B 0,C 180,E1 25089.198,E2 25089.198} C_VEL
LIN {X 0,Y 531.523,Z 917.676,A -85,B 0,C 180,E1 25087.668,E2 25087.668} C_VEL
LIN {X 0,Y 532.469,Z 898.804,A -85,B 0,C 180,E1 25086.19,E2 25086.19} C_VEL
LIN {X 0,Y 533.342,Z 880.351,A -85,B 0,C 180,E1 25084.993,E2 25084.993} C_VEL
LIN {X 0,Y 534.147,Z 861.305,A -85,B 0,C 180,E1 25083.988,E2 25083.988} C_VEL
LIN {X 0,Y 534.913,Z 840.842,A -85,B 0,C 180,E1 25083.136,E2 25083.136} C_VEL
LIN {X 0,Y 535.527,Z 820.424,A -85,B 0,C 180,E1 25082.505,E2 25082.505} C_VEL
LIN {X 0,Y 535.941,Z 799.157,A -85,B 0,C 180,E1 25082.064,E2 25082.064} C_VEL
LIN {X 0,Y 536.325,Z 769.969,A -85,B 0,C 180,E1 25081.616,E2 25081.616} C_VEL
LIN {X 0,Y 540.771,Z 754.624,A -85,B 0,C 180,E1 25080.866,E2 25080.866} C_VEL
LIN {X 0,Y 543.847,Z 746.341,A -85,B 0,C 180,E1 25080.542,E2 25080.542} C_VEL
LIN {X 0,Y 547.424,Z 735.682,A -85,B 0,C 180,E1 25080.091,E2 25080.091} C_VEL
LIN {X 0,Y 553.112,Z 721.979,A -85,B 0,C 180,E1 25079.713,E2 25079.713} C_VEL
LIN {X 0,Y 559.709,Z 706.073,A -85,B 0,C 180,E1 25079.484,E2 25079.484} C_VEL
LIN {X 0,Y 563.562,Z 695.199,A -85,B 0,C 180,E1 25079.391,E2 25079.391} C_VEL
LIN {X 0,Y 566.749,Z 684.396,A -85,B 0,C 180,E1 25079.082,E2 25079.082} C_VEL
LIN {X 0,Y 571.955,Z 664.21,A -85,B 0,C 180,E1 25078.767,E2 25078.767} C_VEL
LIN {X 0,Y 575.604,Z 643.03,A -85,B 0,C 180,E1 25078.506,E2 25078.506} C_VEL
LIN {X 0,Y 578.919,Z 606.468,A -85,B 0,C 180,E1 25078.009,E2 25078.009} C_VEL
LIN {X 0,Y 583.867,Z 614.587,A -85,B 0,C 180,E1 25077.21,E2 25077.21} C_VEL
LIN {X 0,Y 585.431,Z 618.352,A -85,B 0,C 180,E1 25076.667,E2 25076.667} C_VEL
LIN {X 0,Y 585.449,Z 621.153,A -85,B 0,C 180,E1 25076.1,E2 25076.1} C_VEL
LIN {X 0,Y 583.969,Z 623.089,A -85,B 0,C 180,E1 25075.478,E2 25075.478} C_VEL
LIN {X 0,Y 581.428,Z 623.885,A -85,B 0,C 180,E1 25074.94,E2 25074.94} C_VEL
LIN {X 0,Y 577.78,Z 623.589,A -85,B 0,C 180,E1 25074.424,E2 25074.424} C_VEL
LIN {X 0,Y 572.762,Z 621.896,A -85,B 0,C 180,E1 25073.925,E2 25073.925} C_VEL
LIN {X 0,Y 564.15,Z 617.119,A -85,B 0,C 180,E1 25073.065,E2 25073.065} C_VEL
LIN {X 0,Y 556.916,Z 611.052,A -85,B 0,C 180,E1 25072.181,E2 25072.181} C_VEL
LIN {X 0,Y 550.727,Z 603.305,A -85,B 0,C 180,E1 25071.219,E2 25071.219} C_VEL
LIN {X 0,Y 546.115,Z 594.464,A -85,B 0,C 180,E1 25070.26,E2 25070.26} C_VEL
LIN {X 0,Y 542.731,Z 583.548,A -85,B 0,C 180,E1 25069.215,E2 25069.215} C_VEL
LIN {X 0,Y 540.693,Z 570.266,A -85,B 0,C 180,E1 25068.077,E2 25068.077} C_VEL
LIN {X 0,Y 540.185,Z 551.416,A -85,B 0,C 180,E1 25066.631,E2 25066.631} C_VEL
LIN {X 0,Y 542.213,Z 509.34,A -85,B 0,C 180,E1 25063.504,E2 25063.504} C_VEL
LIN {X 0,Y 543.566,Z 481.033,A -85,B 0,C 180,E1 25061.327,E2 25061.327} C_VEL
LIN {X 0,Y 534.602,Z 462.483,A -85,B 0,C 180,E1 25058.796,E2 25058.796} C_VEL
LIN {X 0,Y 530.206,Z 453.699,A -85,B 0,C 180,E1 25057.525,E2 25057.525} C_VEL
LIN {X 0,Y 528.599,Z 450.391,A -85,B 0,C 180,E1 25057.04,E2 25057.04} C_VEL
LIN {X 0,Y 528.473,Z 449.65,A -85,B 0,C 180,E1 25056.952,E2 25056.952} C_VEL
LIN {X 0,Y 528.505,Z 449.652,A -85,B 0,C 180,E1 25053.457,E2 25053.457} C_VEL
LIN {X 0,Y 528.534,Z 449.649,A -85,B 0,C 180,E1 25049.955,E2 25049.955} C_VEL
LIN {X 0,Y 528.505,Z 449.656,A -85,B 0,C 180,E1 25046.512,E2 25046.512} C_VEL
LIN {X 0,Y 528.524,Z 449.652,A -85,B 0,C 180,E1 25043.054,E2 25043.054} C_VEL
LIN {X 0,Y 528.515,Z 449.655,A -85,B 0,C 180,E1 25039.589,E2 25039.589} C_VEL
LIN {X 0,Y 528.521,Z 449.653,A -85,B 0,C 180,E1 25036.146,E2 25036.146} C_VEL
LIN {X 0,Y 528.497,Z 449.656,A -85,B 0,C 180,E1 25032.788,E2 25032.788} C_VEL
LIN {X 0,Y 528.522,Z 449.65,A -85,B 0,C 180,E1 25029.253,E2 25029.253} C_VEL
LIN {X 0,Y 528.499,Z 449.653,A -85,B 0,C 180,E1 25025.863,E2 25025.863} C_VEL
LIN {X 0,Y 528.472,Z 449.655,A -85,B 0,C 180,E1 25022.385,E2 25022.385} C_VEL
LIN {X 0,Y 528.523,Z 449.648,A -85,B 0,C 180,E1 25019.133,E2 25019.133} C_VEL
LIN {X 0,Y 528.472,Z 449.654,A -85,B 0,C 180,E1 25015.768,E2 25015.768} C_VEL
LIN {X 0,Y 528.497,Z 449.644,A -85,B 0,C 180,E1 25012.171,E2 25012.171} C_VEL
LIN {X 0,Y 528.51,Z 449.65,A -85,B 0,C 180,E1 25008.874,E2 25008.874} C_VEL
LIN {X 0,Y 528.477,Z 449.652,A -85,B 0,C 180,E1 25005.426,E2 25005.426} C_VEL
LIN {X 0,Y 528.517,Z 449.644,A -85,B 0,C 180,E1 25002.039,E2 25002.039} C_VEL
LIN {X 0,Y 528.487,Z 449.654,A -85,B 0,C 180,E1 24998.7,E2 24998.7} C_VEL
LIN {X 0,Y 528.502,Z 449.653,A -85,B 0,C 180,E1 24995.285,E2 24995.285} C_VEL
LIN {X 0,Y 528.529,Z 449.648,A -85,B 0,C 180,E1 24991.831,E2 24991.831} C_VEL
LIN {X 0,Y 528.514,Z 449.649,A -85,B 0,C 180,E1 24988.355,E2 24988.355} C_VEL
LIN {X 0,Y 528.522,Z 449.65,A -85,B 0,C 180,E1 24984.893,E2 24984.893} C_VEL
LIN {X 0,Y 528.521,Z 449.65,A -85,B 0,C 180,E1 24981.643,E2 24981.643} C_VEL
LIN {X 0,Y 527.495,Z 449.782,A -85,B 0,C 180,E1 24980.809,E2 24980.809} C_VEL
LIN {X 0,Y 521.105,Z 450.579,A -85,B 0,C 180,E1 24978.463,E2 24978.463} C_VEL
LIN {X 0,Y 520.586,Z 450.64,A -85,B 0,C 180,E1 24977.852,E2 24977.852} C_VEL
LIN {X 0,Y 520.542,Z 450.643,A -85,B 0,C 180,E1 24974.36,E2 24974.36} C_VEL
LIN {X 0,Y 520.556,Z 450.644,A -85,B 0,C 180,E1 24970.772,E2 24970.772} C_VEL
LIN {X 0,Y 520.58,Z 450.642,A -85,B 0,C 180,E1 24967.367,E2 24967.367} C_VEL
LIN {X 0,Y 520.61,Z 450.848,A -85,B 0,C 180,E1 24966.675,E2 24966.675} C_VEL
LIN {X 0,Y 529.175,Z 474.136,A -85,B 0,C 180,E1 24964.006,E2 24964.006} C_VEL
LIN {X 0,Y 528.518,Z 496.182,A -85,B 0,C 180,E1 24962.238,E2 24962.238} C_VEL
LIN {X 0,Y 531.262,Z 511.625,A -85,B 0,C 180,E1 24961.808,E2 24961.808} C_VEL
LIN {X 0,Y 528.767,Z 755.514,A -85,B 0,C 180,E1 24958.184,E2 24958.184} C_VEL
LIN {X 0,Y 528.198,Z 776.56,A -85,B 0,C 180,E1 24957.679,E2 24957.679} C_VEL
LIN {X 0,Y 527.492,Z 797.18,A -85,B 0,C 180,E1 24956.968,E2 24956.968} C_VEL
LIN {X 0,Y 526.677,Z 816.233,A -85,B 0,C 180,E1 24956.109,E2 24956.109} C_VEL
LIN {X 0,Y 525.737,Z 835.318,A -85,B 0,C 180,E1 24955.033,E2 24955.033} C_VEL
LIN {X 0,Y 524.777,Z 853.722,A -85,B 0,C 180,E1 24953.763,E2 24953.763} C_VEL
LIN {X 0,Y 523.798,Z 871.054,A -85,B 0,C 180,E1 24952.325,E2 24952.325} C_VEL
LIN {X 0,Y 522.89,Z 886.944,A -85,B 0,C 180,E1 24950.762,E2 24950.762} C_VEL
LIN {X 0,Y 522.068,Z 902.157,A -85,B 0,C 180,E1 24949,E2 24949} C_VEL
LIN {X 0,Y 521.396,Z 915.523,A -85,B 0,C 180,E1 24947.176,E2 24947.176} C_VEL
LIN {X 0,Y 520.842,Z 928.144,A -85,B 0,C 180,E1 24945.133,E2 24945.133} C_VEL
LIN {X 0,Y 520.438,Z 939.147,A -85,B 0,C 180,E1 24942.989,E2 24942.989} C_VEL
LIN {X 0,Y 520.169,Z 948.254,A -85,B 0,C 180,E1 24940.815,E2 24940.815} C_VEL
LIN {X 0,Y 520.029,Z 955.574,A -85,B 0,C 180,E1 24938.625,E2 24938.625} C_VEL
LIN {X 0,Y 519.95,Z 961.152,A -85,B 0,C 180,E1 24936.403,E2 24936.403} C_VEL
LIN {X 0,Y 519.921,Z 965.019,A -85,B 0,C 180,E1 24934.19,E2 24934.19} C_VEL
LIN {X 0,Y 519.912,Z 967.346,A -85,B 0,C 180,E1 24931.873,E2 24931.873} C_VEL
LIN {X 0,Y 519.903,Z 967.949,A -85,B 0,C 180,E1 24929.669,E2 24929.669} C_VEL
LIN {X 0,Y 519.905,Z 966.991,A -85,B 0,C 180,E1 24927.464,E2 24927.464} C_VEL
LIN {X 0,Y 519.922,Z 964.356,A -85,B 0,C 180,E1 24925.256,E2 24925.256} C_VEL
LIN {X 0,Y 519.955,Z 960.092,A -85,B 0,C 180,E1 24923.041,E2 24923.041} C_VEL
LIN {X 0,Y 520.036,Z 954.112,A -85,B 0,C 180,E1 24920.817,E2 24920.817} C_VEL
LIN {X 0,Y 520.206,Z 946.723,A -85,B 0,C 180,E1 24918.693,E2 24918.693} C_VEL
LIN {X 0,Y 520.499,Z 937.477,A -85,B 0,C 180,E1 24916.559,E2 24916.559} C_VEL
LIN {X 0,Y 520.934,Z 926.093,A -85,B 0,C 180,E1 24914.412,E2 24914.412} C_VEL
LIN {X 0,Y 521.488,Z 913.818,A -85,B 0,C 180,E1 24912.481,E2 24912.481} C_VEL
LIN {X 0,Y 522.179,Z 900.114,A -85,B 0,C 180,E1 24910.654,E2 24910.654} C_VEL
LIN {X 0,Y 523.001,Z 884.921,A -85,B 0,C 180,E1 24908.935,E2 24908.935} C_VEL
LIN {X 0,Y 523.941,Z 868.099,A -85,B 0,C 180,E1 24907.326,E2 24907.326} C_VEL
LIN {X 0,Y 524.951,Z 850.131,A -85,B 0,C 180,E1 24905.885,E2 24905.885} C_VEL
LIN {X 0,Y 525.909,Z 831.952,A -85,B 0,C 180,E1 24904.673,E2 24904.673} C_VEL
LIN {X 0,Y 526.827,Z 812.904,A -85,B 0,C 180,E1 24903.633,E2 24903.633} C_VEL
LIN {X 0,Y 527.68,Z 792.799,A -85,B 0,C 180,E1 24902.767,E2 24902.767} C_VEL
LIN {X 0,Y 528.367,Z 772.075,A -85,B 0,C 180,E1 24902.102,E2 24902.102} C_VEL
LIN {X 0,Y 528.834,Z 751.591,A -85,B 0,C 180,E1 24901.653,E2 24901.653} C_VEL
LIN {X 0,Y 531.122,Z 516.094,A -85,B 0,C 180,E1 24898.162,E2 24898.162} C_VEL
LIN {X 0,Y 526.206,Z 498.051,A -85,B 0,C 180,E1 24897.529,E2 24897.529} C_VEL
LIN {X 0,Y 527.226,Z 473.099,A -85,B 0,C 180,E1 24894.447,E2 24894.447} C_VEL
LIN {X 0,Y 525.262,Z 465.737,A -85,B 0,C 180,E1 24893.355,E2 24893.355} C_VEL
LIN {X 0,Y 520.59,Z 450.646,A -85,B 0,C 180,E1 24890.987,E2 24890.987} C_VEL
LIN {X 0,Y 520.565,Z 450.644,A -85,B 0,C 180,E1 24887.524,E2 24887.524} C_VEL
LIN {X 0,Y 520.563,Z 450.637,A -85,B 0,C 180,E1 24884.052,E2 24884.052} C_VEL
LIN {X 0,Y 520.58,Z 450.638,A -85,B 0,C 180,E1 24880.625,E2 24880.625} C_VEL
LIN {X 0,Y 520.583,Z 450.643,A -85,B 0,C 180,E1 24877.091,E2 24877.091} C_VEL
LIN {X 0,Y 520.577,Z 450.646,A -85,B 0,C 180,E1 24873.584,E2 24873.584} C_VEL
LIN {X 0,Y 520.602,Z 450.802,A -85,B 0,C 180,E1 24871.488,E2 24871.488} C_VEL
LIN {X 0,Y 528.114,Z 472.784,A -85,B 0,C 180,E1 24868.62,E2 24868.62} C_VEL
LIN {X 0,Y 527.2,Z 501.213,A -85,B 0,C 180,E1 24865.802,E2 24865.802} C_VEL
LIN {X 0,Y 525.965,Z 534.319,A -85,B 0,C 180,E1 24862.582,E2 24862.582} C_VEL
LIN {X 0,Y 524.709,Z 570.995,A -85,B 0,C 180,E1 24859.063,E2 24859.063} C_VEL
LIN {X 0,Y 523.684,Z 606.775,A -85,B 0,C 180,E1 24855.674,E2 24855.674} C_VEL
LIN {X 0,Y 523.769,Z 608.409,A -85,B 0,C 180,E1 24855.566,E2 24855.566} C_VEL
LIN {X 0,Y 524.326,Z 614.034,A -85,B 0,C 180,E1 24855.451,E2 24855.451} C_VEL
LIN {X 0,Y 523.047,Z 749.966,A -85,B 0,C 180,E1 24853.355,E2 24853.355} C_VEL
LIN {X 0,Y 522.849,Z 766.903,A -85,B 0,C 180,E1 24852.873,E2 24852.873} C_VEL
LIN {X 0,Y 522.548,Z 782.501,A -85,B 0,C 180,E1 24852.207,E2 24852.207} C_VEL
LIN {X 0,Y 522.177,Z 797.883,A -85,B 0,C 180,E1 24851.319,E2 24851.319} C_VEL
LIN {X 0,Y 521.78,Z 811.177,A -85,B 0,C 180,E1 24850.322,E2 24850.322} C_VEL
LIN {X 0,Y 521.362,Z 824.149,A -85,B 0,C 180,E1 24849.104,E2 24849.104} C_VEL
LIN {X 0,Y 521.008,Z 834.961,A -85,B 0,C 180,E1 24847.831,E2 24847.831} C_VEL
LIN {X 0,Y 520.702,Z 844.819,A -85,B 0,C 180,E1 24846.395,E2 24846.395} C_VEL
LIN {X 0,Y 520.471,Z 853.258,A -85,B 0,C 180,E1 24844.849,E2 24844.849} C_VEL
LIN {X 0,Y 520.303,Z 860.135,A -85,B 0,C 180,E1 24843.195,E2 24843.195} C_VEL
LIN {X 0,Y 520.204,Z 865.265,A -85,B 0,C 180,E1 24841.542,E2 24841.542} C_VEL
LIN {X 0,Y 520.159,Z 868.885,A -85,B 0,C 180,E1 24839.78,E2 24839.78} C_VEL
LIN {X 0,Y 520.142,Z 870.778,A -85,B 0,C 180,E1 24838.017,E2 24838.017} C_VEL
LIN {X 0,Y 520.149,Z 871.076,A -85,B 0,C 180,E1 24836.253,E2 24836.253} C_VEL
LIN {X 0,Y 520.184,Z 869.601,A -85,B 0,C 180,E1 24834.485,E2 24834.485} C_VEL
LIN {X 0,Y 520.245,Z 866.75,A -85,B 0,C 180,E1 24832.824,E2 24832.824} C_VEL
LIN {X 0,Y 520.373,Z 861.91,A -85,B 0,C 180,E1 24831.047,E2 24831.047} C_VEL
LIN {X 0,Y 520.568,Z 855.46,A -85,B 0,C 180,E1 24829.375,E2 24829.375} C_VEL
LIN {X 0,Y 520.811,Z 847.595,A -85,B 0,C 180,E1 24827.809,E2 24827.809} C_VEL
LIN {X 0,Y 521.139,Z 838.205,A -85,B 0,C 180,E1 24826.35,E2 24826.35} C_VEL
LIN {X 0,Y 521.537,Z 827.38,A -85,B 0,C 180,E1 24825.001,E2 24825.001} C_VEL
LIN {X 0,Y 521.936,Z 815.436,A -85,B 0,C 180,E1 24823.816,E2 24823.816} C_VEL
LIN {X 0,Y 522.357,Z 801.864,A -85,B 0,C 180,E1 24822.741,E2 24822.741} C_VEL
LIN {X 0,Y 522.678,Z 787.967,A -85,B 0,C 180,E1 24821.889,E2 24821.889} C_VEL
LIN {X 0,Y 522.946,Z 773.208,A -85,B 0,C 180,E1 24821.206,E2 24821.206} C_VEL
LIN {X 0,Y 523.091,Z 757.653,A -85,B 0,C 180,E1 24820.701,E2 24820.701} C_VEL
LIN {X 0,Y 523.167,Z 737.389,A -85,B 0,C 180,E1 24820.319,E2 24820.319} C_VEL
LIN {X 0,Y 524.72,Z 635.739,A -85,B 0,C 180,E1 24818.62,E2 24818.62} C_VEL
LIN {X 0,Y 525.183,Z 616.636,A -85,B 0,C 180,E1 24818.266,E2 24818.266} C_VEL
LIN {X 0,Y 526.245,Z 612.969,A -85,B 0,C 180,E1 24817.961,E2 24817.961} C_VEL
LIN {X 0,Y 528.976,Z 576.928,A -85,B 0,C 180,E1 24814.171,E2 24814.171} C_VEL
LIN {X 0,Y 532.598,Z 544.225,A -85,B 0,C 180,E1 24810.537,E2 24810.537} C_VEL
LIN {X 0,Y 536.947,Z 517.154,A -85,B 0,C 180,E1 24807.316,E2 24807.316} C_VEL
LIN {X 0,Y 539.797,Z 503.84,A -85,B 0,C 180,E1 24805.602,E2 24805.602} C_VEL
LIN {X 0,Y 542.129,Z 493.491,A -85,B 0,C 180,E1 24804.063,E2 24804.063} C_VEL
LIN {X 0,Y 541.135,Z 489.274,A -85,B 0,C 180,E1 24802.563,E2 24802.563} C_VEL
LIN {X 0,Y 540.899,Z 487.043,A -85,B 0,C 180,E1 24801.333,E2 24801.333} C_VEL
LIN {X 0,Y 541.017,Z 486.776,A -85,B 0,C 180,E1 24799.918,E2 24799.918} C_VEL
LIN {X 0,Y 541.763,Z 488.099,A -85,B 0,C 180,E1 24798.851,E2 24798.851} C_VEL
LIN {X 0,Y 541.858,Z 488.676,A -85,B 0,C 180,E1 24798.655,E2 24798.655} C_VEL
LIN {X 0,Y 537.123,Z 502.204,A -85,B 0,C 180,E1 24797.254,E2 24797.254} C_VEL
LIN {X 0,Y 533.24,Z 519.536,A -85,B 0,C 180,E1 24795.672,E2 24795.672} C_VEL
LIN {X 0,Y 530.214,Z 542.521,A -85,B 0,C 180,E1 24793.795,E2 24793.795} C_VEL
LIN {X 0,Y 529.653,Z 561.633,A -85,B 0,C 180,E1 24792.269,E2 24792.269} C_VEL
LIN {X 0,Y 531.01,Z 576.368,A -85,B 0,C 180,E1 24791.06,E2 24791.06} C_VEL
LIN {X 0,Y 534.333,Z 589.791,A -85,B 0,C 180,E1 24789.897,E2 24789.897} C_VEL
LIN {X 0,Y 539.018,Z 600.558,A -85,B 0,C 180,E1 24788.908,E2 24788.908} C_VEL
LIN {X 0,Y 545.392,Z 610.095,A -85,B 0,C 180,E1 24787.972,E2 24787.972} C_VEL
LIN {X 0,Y 553.07,Z 618.119,A -85,B 0,C 180,E1 24787.132,E2 24787.132} C_VEL
LIN {X 0,Y 562.256,Z 624.938,A -85,B 0,C 180,E1 24786.335,E2 24786.335} C_VEL
LIN {X 0,Y 571.143,Z 629.535,A -85,B 0,C 180,E1 24785.68,E2 24785.68} C_VEL
LIN {X 0,Y 576.04,Z 630.872,A -85,B 0,C 180,E1 24785.189,E2 24785.189} C_VEL
LIN {X 0,Y 579.74,Z 630.892,A -85,B 0,C 180,E1 24784.648,E2 24784.648} C_VEL
LIN {X 0,Y 582.344,Z 629.693,A -85,B 0,C 180,E1 24784.038,E2 24784.038} C_VEL
LIN {X 0,Y 583.456,Z 627.391,A -85,B 0,C 180,E1 24783.406,E2 24783.406} C_VEL
LIN {X 0,Y 582.954,Z 624.127,A -85,B 0,C 180,E1 24782.815,E2 24782.815} C_VEL
LIN {X 0,Y 581.746,Z 621.789,A -85,B 0,C 180,E1 24782.465,E2 24782.465} C_VEL
LIN {X 0,Y 578.374,Z 642.096,A -85,B 0,C 180,E1 24782.266,E2 24782.266} C_VEL
LIN {X 0,Y 573.134,Z 662.132,A -85,B 0,C 180,E1 24782.064,E2 24782.064} C_VEL
LIN {X 0,Y 566.067,Z 682.623,A -85,B 0,C 180,E1 24781.761,E2 24781.761} C_VEL
LIN {X 0,Y 561.627,Z 694.756,A -85,B 0,C 180,E1 24781.442,E2 24781.442} C_VEL
LIN {X 0,Y 560.86,Z 696.932,A -85,B 0,C 180,E1 24781.37,E2 24781.37} C_VEL
LIN {X 0,Y 552.568,Z 713.515,A -85,B 0,C 180,E1 24781.143,E2 24781.143} C_VEL
LIN {X 0,Y 544.935,Z 728.272,A -85,B 0,C 180,E1 24780.751,E2 24780.751} C_VEL
LIN {X 0,Y 539.362,Z 741.065,A -85,B 0,C 180,E1 24780.247,E2 24780.247} C_VEL
LIN {X 0,Y 536.664,Z 748.914,A -85,B 0,C 180,E1 24779.88,E2 24779.88} C_VEL
LIN {X 0,Y 532.623,Z 759.443,A -85,B 0,C 180,E1 24779.4,E2 24779.4} C_VEL
LIN {X 0,Y 529.113,Z 772.85,A -85,B 0,C 180,E1 24778.725,E2 24778.725} C_VEL
LIN {X 0,Y 528.724,Z 807.903,A -85,B 0,C 180,E1 24778.184,E2 24778.184} C_VEL
LIN {X 0,Y 528.141,Z 829.167,A -85,B 0,C 180,E1 24777.65,E2 24777.65} C_VEL
LIN {X 0,Y 527.429,Z 849.035,A -85,B 0,C 180,E1 24776.942,E2 24776.942} C_VEL
LIN {X 0,Y 526.56,Z 868.88,A -85,B 0,C 180,E1 24776.017,E2 24776.017} C_VEL
LIN {X 0,Y 525.597,Z 888.06,A -85,B 0,C 180,E1 24774.905,E2 24774.905} C_VEL
LIN {X 0,Y 524.603,Z 906.467,A -85,B 0,C 180,E1 24773.594,E2 24773.594} C_VEL
LIN {X 0,Y 523.629,Z 924.034,A -85,B 0,C 180,E1 24772.097,E2 24772.097} C_VEL
LIN {X 0,Y 522.736,Z 939.85,A -85,B 0,C 180,E1 24770.49,E2 24770.49} C_VEL
LIN {X 0,Y 521.997,Z 953.495,A -85,B 0,C 180,E1 24768.875,E2 24768.875} C_VEL
LIN {X 0,Y 521.316,Z 967.324,A -85,B 0,C 180,E1 24766.95,E2 24766.95} C_VEL
LIN {X 0,Y 520.812,Z 978.808,A -85,B 0,C 180,E1 24765.059,E2 24765.059} C_VEL
LIN {X 0,Y 520.414,Z 989.848,A -85,B 0,C 180,E1 24762.878,E2 24762.878} C_VEL
LIN {X 0,Y 520.162,Z 998.691,A -85,B 0,C 180,E1 24760.747,E2 24760.747} C_VEL
